C05497=1160.781,162.301,-57.931,-178.413,6.811,148.793
C05498=1160.776,162.550,-57.953,-178.410,6.813,148.793
C05499=1160.772,162.799,-57.975,-178.407,6.815,148.793
C05500=1160.767,163.048,-57.997,-178.404,6.817,148.792
C05501=1160.762,163.296,-58.018,-178.401,6.819,148.792
C05502=1160.758,163.546,-58.040,-178.399,6.821,148.792
C05503=1160.753,163.794,-58.062,-178.396,6.823,148.791
C05504=1160.749,164.044,-58.084,-178.394,6.824,148.791
C05505=1160.744,164.292,-58.106,-178.390,6.827,148.791
C05506=1160.740,164.542,-58.128,-178.388,6.829,148.790
C05507=1160.735,164.790,-58.149,-178.385,6.831,148.790
C05508=1160.731,165.040,-58.172,-178.382,6.832,148.790
C05509=1160.725,165.289,-58.194,-178.380,6.834,148.789
C05510=1160.721,165.538,-58.216,-178.377,6.836,148.789
C05511=1160.716,165.787,-58.238,-178.374,6.839,148.789
C05512=1160.712,166.036,-58.260,-178.371,6.840,148.788
C05513=1160.707,166.285,-58.281,-178.369,6.842,148.788
C05514=1160.703,166.534,-58.303,-178.366,6.844,148.788
C05515=1160.698,166.783,-58.325,-178.363,6.846,148.787
C05516=1160.692,167.032,-58.347,-178.360,6.848,148.787
C05517=1160.688,167.281,-58.369,-178.358,6.850,148.787
C05518=1160.683,167.529,-58.392,-178.355,6.852,148.786
C05519=1160.679,167.778,-58.414,-178.352,6.854,148.786
C05520=1160.675,168.028,-58.436,-178.350,6.856,148.786
C05521=1160.669,168.276,-58.458,-178.346,6.858,148.785
C05522=1160.665,168.526,-58.480,-178.344,6.860,148.785
C05523=1160.660,168.774,-58.502,-178.342,6.862,148.785
C05524=1160.656,169.023,-58.525,-178.339,6.864,148.784
C05525=1160.650,169.272,-58.547,-178.336,6.865,148.784
C05526=1160.646,169.521,-58.569,-178.333,6.868,148.784
C05527=1160.641,169.770,-58.591,-178.330,6.870,148.783
C05528=1160.637,170.019,-58.613,-178.328,6.872,148.783
C05529=1160.632,170.268,-58.636,-178.325,6.874,148.783
C05530=1160.627,170.517,-58.658,-178.322,6.876,148.782
C05531=1160.623,170.766,-58.679,-178.319,6.878,148.782
C05532=1160.618,171.015,-58.702,-178.317,6.880,148.782
C05533=1160.614,171.264,-58.725,-178.314,6.881,148.781
C05534=1160.609,171.513,-58.746,-178.312,6.884,148.781
C05535=1160.604,171.762,-58.769,-178.308,6.886,148.781
C05536=1160.599,172.010,-58.792,-178.306,6.888,148.780
C05537=1160.595,172.260,-58.814,-178.303,6.890,148.780
C05538=1160.590,172.509,-58.836,-178.300,6.891,148.780
C05539=1160.585,172.757,-58.859,-178.297,6.894,148.779
C05540=1160.581,173.007,-58.881,-178.295,6.896,148.779
C05541=1160.575,173.256,-58.903,-178.292,6.898,148.779
C05542=1160.571,173.504,-58.926,-178.290,6.899,148.779
C05543=1160.567,173.754,-58.948,-178.286,6.902,148.778
C05544=1160.562,174.002,-58.971,-178.284,6.904,148.778
C05545=1160.558,174.252,-58.993,-178.281,6.906,148.778
C05546=1160.553,174.501,-59.016,-178.279,6.908,148.777
C05547=1160.548,174.749,-59.038,-178.275,6.910,148.777
C05548=1160.544,174.998,-59.061,-178.273,6.912,148.777
C05549=1160.539,175.248,-59.083,-178.271,6.914,148.776
C05550=1160.534,175.496,-59.105,-178.268,6.916,148.776
C05551=1160.529,175.745,-59.128,-178.265,6.918,148.776
C05552=1160.525,175.995,-59.150,-178.262,6.920,148.775
C05553=1160.520,176.243,-59.173,-178.259,6.922,148.775
C05554=1160.516,176.492,-59.196,-178.256,6.925,148.775
C05555=1160.511,176.741,-59.219,-178.254,6.927,148.775
C05556=1160.506,176.989,-59.241,-178.251,6.928,148.774
C05557=1160.501,177.239,-59.264,-178.248,6.930,148.774
C05558=1160.497,177.488,-59.287,-178.246,6.933,148.774
C05559=1160.492,177.737,-59.309,-178.243,6.935,148.773
C05560=1160.488,177.985,-59.332,-178.240,6.936,148.773
C05561=1160.483,178.234,-59.355,-178.237,6.938,148.773
C05562=1160.479,178.484,-59.377,-178.235,6.941,148.772
C05563=1160.474,178.732,-59.400,-178.232,6.943,148.772
C05564=1160.470,178.981,-59.423,-178.229,6.945,148.772
C05565=1160.465,179.230,-59.445,-178.226,6.947,148.771
C05566=1160.461,179.479,-59.468,-178.224,6.949,148.771
C05567=1160.455,179.727,-59.491,-178.221,6.951,148.771
C05568=1160.450,179.977,-59.514,-178.218,6.953,148.771
C05569=1160.446,180.226,-59.537,-178.215,6.955,148.770
C05570=1160.442,180.475,-59.560,-178.213,6.958,148.770
C05571=1160.437,180.723,-59.582,-178.210,6.959,148.770
C05572=1160.432,180.973,-59.605,-178.207,6.962,148.769
C05573=1160.427,181.222,-59.628,-178.204,6.964,148.769
C05574=1160.423,181.470,-59.651,-178.202,6.966,148.769
C05575=1160.419,181.719,-59.674,-178.199,6.968,148.768
C05576=1160.414,181.968,-59.696,-178.196,6.970,148.768
C05577=1160.409,182.217,-59.719,-178.193,6.972,148.768
C05578=1160.404,182.466,-59.743,-178.191,6.975,148.768
C05579=1160.401,182.715,-59.766,-178.188,6.976,148.767
C05580=1160.396,182.964,-59.789,-178.185,6.978,148.767
C05581=1160.391,183.213,-59.812,-178.183,6.980,148.767
C05582=1160.386,183.461,-59.834,-178.180,6.983,148.766
C05583=1160.381,183.731,-59.860,-178.177,6.985,148.766
C05584=1160.376,184.000,-59.885,-178.174,6.987,148.766
C05585=1160.372,184.271,-59.910,-178.171,6.990,148.765
C05586=1160.367,184.540,-59.935,-178.168,6.992,148.765
C05587=1160.361,184.789,-59.958,-178.165,6.994,148.765
C05588=1160.357,185.038,-59.981,-178.162,6.996,148.765
C05589=1160.353,185.286,-60.004,-178.160,6.998,148.764
C05590=1160.348,185.535,-60.027,-178.157,7.001,148.764
C05591=1160.343,185.784,-60.050,-178.154,7.003,148.764
C05592=1160.339,186.033,-60.074,-178.152,7.004,148.763
C05593=1160.335,186.282,-60.097,-178.148,7.007,148.763
C05594=1160.330,186.531,-60.120,-178.146,7.009,148.763
C05595=1160.325,186.780,-60.143,-178.143,7.011,148.763
C05596=1160.320,187.029,-60.166,-178.140,7.013,148.762
C05597=1160.315,187.278,-60.190,-178.138,7.016,148.762
C05598=1160.311,187.526,-60.212,-178.135,7.017,148.762
C05599=1160.307,187.775,-60.236,-178.132,7.020,148.761
C05600=1160.302,188.024,-60.259,-178.130,7.022,148.761
C05601=1160.297,188.273,-60.282,-178.127,7.024,148.761
C05602=1160.292,188.522,-60.306,-178.124,7.026,148.761
C05603=1160.288,188.771,-60.330,-178.122,7.028,148.760
C05604=1160.283,189.020,-60.353,-178.119,7.030,148.760
C05605=1160.279,189.269,-60.377,-178.116,7.033,148.760
C05606=1160.275,189.518,-60.399,-178.114,7.035,148.760
C05607=1160.270,189.767,-60.423,-178.110,7.037,148.759
C05608=1160.265,190.015,-60.446,-178.108,7.039,148.759
C05609=1160.260,190.263,-60.470,-178.105,7.041,148.759
C05610=1160.256,190.512,-60.493,-178.102,7.044,148.758
C05611=1160.251,190.762,-60.517,-178.099,7.046,148.758
C05612=1160.246,191.011,-60.540,-178.097,7.048,148.758
C05613=1160.241,191.260,-60.563,-178.094,7.050,148.758
C05614=1160.237,191.508,-60.587,-178.091,7.052,148.757
C05615=1160.232,191.757,-60.611,-178.088,7.055,148.757
C05616=1160.228,192.006,-60.634,-178.086,7.057,148.757
C05617=1160.223,192.254,-60.658,-178.083,7.058,148.756
C05618=1160.219,192.504,-60.681,-178.080,7.061,148.756
C05619=1160.214,192.753,-60.705,-178.078,7.063,148.756
C05620=1160.210,193.001,-60.729,-178.075,7.065,148.756
C05621=1160.205,193.250,-60.752,-178.072,7.068,148.756
C05622=1160.200,193.499,-60.776,-178.069,7.070,148.755
C05623=1160.196,193.747,-60.800,-178.067,7.073,148.755
C05624=1160.191,193.996,-60.823,-178.064,7.074,148.755
C05625=1160.187,194.246,-60.847,-178.061,7.076,148.754
C05626=1160.183,194.495,-60.871,-178.059,7.079,148.754
C05627=1160.178,194.744,-60.894,-178.056,7.081,148.754
C05628=1160.173,194.992,-60.918,-178.053,7.083,148.754
C05629=1160.169,195.241,-60.942,-178.050,7.085,148.753
C05630=1160.164,195.490,-60.965,-178.047,7.088,148.753
C05631=1160.160,195.739,-60.989,-178.045,7.090,148.753
C05632=1160.155,195.988,-61.012,-178.042,7.092,148.753
C05633=1160.150,196.236,-61.037,-178.039,7.094,148.752
C05634=1160.145,196.485,-61.060,-178.037,7.097,148.752
C05635=1160.141,196.734,-61.085,-178.034,7.099,148.752
C05636=1160.136,196.983,-61.108,-178.031,7.101,148.752
C05637=1160.132,197.231,-61.132,-178.029,7.103,148.751
C05638=1160.128,197.480,-61.156,-178.025,7.106,148.751
C05639=1160.123,197.729,-61.180,-178.023,7.108,148.751
C05640=1160.119,197.978,-61.204,-178.020,7.110,148.751
C05641=1160.113,198.227,-61.228,-178.018,7.112,148.750
C05642=1160.109,198.475,-61.252,-178.014,7.115,148.750
C05643=1160.104,198.725,-61.275,-178.012,7.117,148.750
C05644=1160.100,198.973,-61.299,-178.010,7.119,148.750
C05645=1160.095,199.221,-61.323,-178.006,7.121,148.749
C05646=1160.091,199.471,-61.348,-178.004,7.124,148.749
C05647=1160.086,199.720,-61.372,-178.001,7.126,148.749
C05648=1160.082,199.968,-61.396,-177.998,7.128,148.749
C05649=1160.077,200.217,-61.419,-177.995,7.131,148.748
C05650=1160.073,200.466,-61.443,-177.993,7.133,148.748
C05651=1160.068,200.714,-61.468,-177.990,7.136,148.748
C05652=1160.063,200.964,-61.492,-177.987,7.137,148.748
C05653=1160.059,201.213,-61.516,-177.985,7.139,148.747
C05654=1160.055,201.461,-61.540,-177.982,7.142,148.747
C05655=1160.050,201.710,-61.565,-177.979,7.144,148.747
C05656=1160.045,201.959,-61.588,-177.976,7.147,148.747
C05657=1160.041,202.208,-61.612,-177.974,7.148,148.746
C05658=1160.036,202.457,-61.637,-177.971,7.151,148.746
C05659=1160.032,202.705,-61.661,-177.968,7.153,148.746
C05660=1160.027,202.953,-61.685,-177.965,7.156,148.746
C05661=1160.022,203.203,-61.709,-177.963,7.158,148.745
C05662=1160.018,203.452,-61.734,-177.960,7.161,148.745
C05663=1160.014,203.700,-61.758,-177.957,7.163,148.745
C05664=1160.008,203.949,-61.782,-177.954,7.165,148.745
C05665=1160.005,204.198,-61.807,-177.952,7.167,148.745
C05666=1160.000,204.446,-61.831,-177.949,7.169,148.744
C05667=1159.995,204.695,-61.855,-177.946,7.172,148.744
C05668=1159.991,204.944,-61.880,-177.944,7.174,148.744
C05669=1159.986,205.193,-61.905,-177.941,7.177,148.744
C05670=1159.981,205.442,-61.928,-177.938,7.178,148.743
C05671=1159.977,205.690,-61.952,-177.935,7.181,148.743
C05672=1159.972,205.939,-61.977,-177.933,7.183,148.743
C05673=1159.968,206.188,-62.001,-177.930,7.186,148.743
C05674=1159.963,206.437,-62.026,-177.927,7.188,148.742
C05675=1159.959,206.685,-62.050,-177.925,7.191,148.742
C05676=1159.954,206.935,-62.075,-177.922,7.192,148.742
C05677=1159.950,207.183,-62.099,-177.919,7.195,148.742
C05678=1159.945,207.432,-62.124,-177.916,7.197,148.742
C05679=1159.941,207.681,-62.148,-177.914,7.200,148.741
C05680=1159.936,207.929,-62.173,-177.911,7.202,148.741
C05681=1159.932,208.178,-62.198,-177.908,7.205,148.741
C05682=1159.926,208.426,-62.222,-177.905,7.207,148.741
C05683=1159.923,208.675,-62.247,-177.903,7.210,148.741
C05684=1159.917,208.924,-62.271,-177.900,7.211,148.740
C05685=1159.914,209.173,-62.296,-177.897,7.214,148.740
C05686=1159.909,209.422,-62.320,-177.895,7.216,148.740
C05687=1159.903,209.692,-62.347,-177.892,7.219,148.740
C05688=1159.899,209.963,-62.374,-177.889,7.221,148.739
C05689=1159.894,210.233,-62.401,-177.885,7.224,148.739
C05690=1159.889,210.504,-62.428,-177.882,7.227,148.739
C05691=1159.885,210.753,-62.452,-177.880,7.229,148.739
C05692=1159.880,211.001,-62.477,-177.877,7.232,148.739
C05693=1159.876,211.250,-62.501,-177.874,7.233,148.738
C05694=1159.871,211.498,-62.527,-177.872,7.236,148.738
C05695=1159.866,211.748,-62.552,-177.869,7.238,148.738
C05696=1159.862,211.996,-62.576,-177.866,7.241,148.738
C05697=1159.857,212.244,-62.601,-177.863,7.243,148.737
C05698=1159.853,212.494,-62.626,-177.861,7.246,148.737
C05699=1159.848,212.742,-62.650,-177.858,7.248,148.737
C05700=1159.844,212.992,-62.675,-177.855,7.251,148.737
C05701=1159.839,213.240,-62.701,-177.852,7.253,148.737
C05702=1159.835,213.488,-62.725,-177.850,7.255,148.736
C05703=1159.830,213.738,-62.750,-177.847,7.258,148.736
C05704=1159.825,213.986,-62.775,-177.844,7.260,148.736
C05705=1159.821,214.235,-62.800,-177.842,7.263,148.736
C05706=1159.817,214.483,-62.825,-177.839,7.265,148.735
C05707=1159.812,214.732,-62.850,-177.836,7.268,148.735
C05708=1159.808,214.981,-62.874,-177.833,7.269,148.735
C05709=1159.803,215.230,-62.900,-177.831,7.272,148.735
C05710=1159.798,215.478,-62.924,-177.828,7.275,148.735
C05711=1159.794,215.727,-62.950,-177.825,7.277,148.735
C05712=1159.790,215.976,-62.974,-177.822,7.280,148.734
C05713=1159.785,216.224,-63.000,-177.820,7.282,148.734
C05714=1159.780,216.473,-63.025,-177.817,7.285,148.734
C05715=1159.776,216.722,-63.050,-177.814,7.286,148.734
C05716=1159.772,216.970,-63.075,-177.812,7.289,148.734
C05717=1159.767,217.219,-63.100,-177.809,7.291,148.733
C05718=1159.762,217.468,-63.125,-177.806,7.294,148.733
C05719=1159.758,217.717,-63.151,-177.803,7.297,148.733
C05720=1159.753,217.965,-63.175,-177.801,7.299,148.733
C05721=1159.750,218.214,-63.201,-177.798,7.302,148.733
C05722=1159.744,218.463,-63.225,-177.795,7.303,148.732
C05723=1159.740,218.711,-63.251,-177.792,7.306,148.732
C05724=1159.736,218.960,-63.277,-177.790,7.309,148.732
C05725=1159.731,219.209,-63.301,-177.787,7.311,148.732
C05726=1159.727,219.458,-63.327,-177.784,7.314,148.732
C05727=1159.722,219.705,-63.352,-177.781,7.316,148.731
C05728=1159.718,219.955,-63.377,-177.779,7.319,148.731
C05729=1159.713,220.203,-63.402,-177.776,7.322,148.731
C05730=1159.709,220.452,-63.428,-177.773,7.323,148.731
C05731=1159.704,220.701,-63.453,-177.770,7.326,148.731
C05732=1159.700,220.949,-63.478,-177.768,7.328,148.730
C05733=1159.695,221.198,-63.504,-177.765,7.331,148.730
C05734=1159.690,221.446,-63.530,-177.762,7.334,148.730
C05735=1159.686,221.696,-63.555,-177.760,7.336,148.730
C05736=1159.682,221.944,-63.580,-177.757,7.339,148.730
C05737=1159.677,222.193,-63.606,-177.754,7.341,148.729
C05738=1159.673,222.441,-63.632,-177.751,7.343,148.729
C05739=1159.668,222.690,-63.656,-177.749,7.346,148.729
C05740=1159.663,222.939,-63.682,-177.746,7.348,148.729
C05741=1159.659,223.188,-63.708,-177.743,7.351,148.729
C05742=1159.654,223.436,-63.733,-177.741,7.353,148.729
C05743=1159.650,223.685,-63.759,-177.738,7.356,148.728
C05744=1159.646,223.933,-63.785,-177.735,7.359,148.728
C05745=1159.641,224.182,-63.809,-177.733,7.361,148.728
C05746=1159.636,224.431,-63.835,-177.729,7.363,148.728
C05747=1159.632,224.680,-63.861,-177.727,7.366,148.728
C05748=1159.627,224.928,-63.886,-177.724,7.368,148.728
C05749=1159.623,225.177,-63.912,-177.721,7.371,148.727
C05750=1159.619,225.425,-63.938,-177.718,7.374,148.727
C05751=1159.614,225.674,-63.963,-177.716,7.376,148.727
C05752=1159.610,225.922,-63.989,-177.713,7.379,148.727
C05753=1159.606,226.171,-64.015,-177.711,7.381,148.727
C05754=1159.601,226.420,-64.040,-177.708,7.383,148.727
C05755=1159.597,226.668,-64.066,-177.705,7.386,148.726
C05756=1159.592,226.917,-64.092,-177.703,7.389,148.726
C05757=1159.587,227.166,-64.118,-177.699,7.391,148.726
C05758=1159.583,227.414,-64.143,-177.697,7.394,148.726
C05759=1159.578,227.663,-64.169,-177.694,7.396,148.726
C05760=1159.574,227.912,-64.195,-177.691,7.399,148.726
C05761=1159.570,228.161,-64.220,-177.688,7.402,148.725
C05762=1159.565,228.409,-64.246,-177.686,7.404,148.725
C05763=1159.560,228.658,-64.272,-177.683,7.406,148.725
C05764=1159.556,228.906,-64.299,-177.680,7.409,148.725
C05765=1159.552,229.155,-64.324,-177.678,7.412,148.725
C05766=1159.547,229.403,-64.350,-177.675,7.414,148.725
C05767=1159.543,229.652,-64.375,-177.672,7.417,148.724
C05768=1159.538,229.901,-64.402,-177.670,7.419,148.724
C05769=1159.534,230.150,-64.428,-177.667,7.422,148.724
C05770=1159.530,230.398,-64.454,-177.664,7.425,148.724
C05771=1159.525,230.646,-64.479,-177.662,7.427,148.724
C05772=1159.520,230.895,-64.506,-177.659,7.430,148.724
C05773=1159.516,231.144,-64.532,-177.656,7.432,148.723
C05774=1159.512,231.393,-64.557,-177.653,7.434,148.723
C05775=1159.508,231.641,-64.584,-177.651,7.437,148.723
C05776=1159.502,231.889,-64.610,-177.648,7.440,148.723
C05777=1159.498,232.138,-64.635,-177.645,7.443,148.723
C05778=1159.494,232.386,-64.662,-177.642,7.445,148.723
C05779=1159.489,232.635,-64.688,-177.640,7.448,148.723
C05780=1159.485,232.884,-64.714,-177.636,7.451,148.722
C05781=1159.481,233.132,-64.741,-177.634,7.453,148.722
C05782=1159.475,233.381,-64.766,-177.631,7.456,148.722
C05783=1159.471,233.630,-64.792,-177.629,7.459,148.722
C05784=1159.467,233.878,-64.819,-177.626,7.460,148.722
C05785=1159.462,234.127,-64.845,-177.623,7.463,148.722
C05786=1159.458,234.376,-64.871,-177.620,7.466,148.722
C05787=1159.454,234.624,-64.897,-177.618,7.469,148.722
C05788=1159.449,234.873,-64.924,-177.615,7.471,148.721
C05789=1159.445,235.121,-64.950,-177.612,7.474,148.721
C05790=1159.440,235.370,-64.976,-177.609,7.477,148.721
C05791=1159.436,235.641,-65.005,-177.606,7.479,148.721
C05792=1159.431,235.913,-65.033,-177.603,7.482,148.721
C05793=1159.426,236.185,-65.063,-177.601,7.485,148.721
C05794=1159.421,236.457,-65.091,-177.597,7.488,148.720
C05795=1159.417,236.705,-65.118,-177.595,7.491,148.720
C05796=1159.413,236.954,-65.144,-177.592,7.493,148.720
C05797=1159.407,237.202,-65.170,-177.590,7.496,148.720
C05798=1159.403,237.450,-65.197,-177.586,7.499,148.720
C05799=1159.398,237.699,-65.223,-177.584,7.502,148.720
C05800=1159.394,237.947,-65.249,-177.581,7.504,148.720
C05801=1159.389,238.197,-65.276,-177.579,7.507,148.720
C05802=1159.386,238.445,-65.302,-177.576,7.510,148.719
C05803=1159.381,238.693,-65.329,-177.573,7.512,148.719
C05804=1159.377,238.942,-65.355,-177.570,7.514,148.719
C05805=1159.372,239.191,-65.382,-177.568,7.517,148.719
C05806=1159.368,239.439,-65.409,-177.565,7.520,148.719
C05807=1159.363,239.688,-65.435,-177.562,7.523,148.719
C05808=1159.358,239.936,-65.462,-177.559,7.525,148.718
C05809=1159.355,240.185,-65.488,-177.557,7.528,148.718
C05810=1159.350,240.434,-65.515,-177.554,7.531,148.718
C05811=1159.346,240.682,-65.541,-177.551,7.534,148.718
C05812=1159.341,240.930,-65.568,-177.548,7.535,148.718
C05813=1159.337,241.179,-65.595,-177.546,7.538,148.718
C05814=1159.332,241.428,-65.621,-177.543,7.541,148.718
C05815=1159.327,241.676,-65.648,-177.540,7.544,148.718
C05816=1159.324,241.924,-65.675,-177.538,7.546,148.718
C05817=1159.319,242.173,-65.702,-177.535,7.549,148.718
C05818=1159.314,242.421,-65.729,-177.532,7.552,148.717
C05819=1159.310,242.670,-65.755,-177.529,7.555,148.717
C05820=1159.305,242.919,-65.782,-177.527,7.557,148.717
C05821=1159.301,243.167,-65.809,-177.524,7.560,148.717
C05822=1159.297,243.415,-65.835,-177.521,7.563,148.717
C05823=1159.293,243.664,-65.863,-177.519,7.566,148.717
C05824=1159.288,243.913,-65.890,-177.515,7.568,148.717
C05825=1159.284,244.161,-65.916,-177.513,7.571,148.716
C05826=1159.279,244.410,-65.943,-177.510,7.574,148.716
C05827=1159.275,244.658,-65.970,-177.508,7.576,148.716
C05828=1159.271,244.907,-65.996,-177.505,7.579,148.716
C05829=1159.266,245.155,-66.023,-177.503,7.582,148.716
C05830=1159.261,245.404,-66.050,-177.500,7.584,148.716
C05831=1159.257,245.652,-66.077,-177.497,7.587,148.716
C05832=1159.253,245.901,-66.104,-177.494,7.590,148.716
C05833=1159.249,246.150,-66.131,-177.491,7.593,148.716
C05834=1159.244,246.398,-66.158,-177.489,7.595,148.716
C05835=1159.239,246.647,-66.185,-177.486,7.598,148.715
C05836=1159.235,246.895,-66.213,-177.483,7.601,148.715
C05837=1159.231,247.143,-66.239,-177.480,7.604,148.715
C05838=1159.226,247.391,-66.266,-177.477,7.607,148.715
C05839=1159.222,247.640,-66.294,-177.475,7.609,148.715
C05840=1159.218,247.889,-66.321,-177.473,7.612,148.715
C05841=1159.213,248.138,-66.348,-177.470,7.615,148.715
C05842=1159.208,248.386,-66.375,-177.467,7.618,148.715
C05843=1159.204,248.634,-66.402,-177.464,7.620,148.715
C05844=1159.200,248.883,-66.429,-177.462,7.623,148.715
C05845=1159.195,249.131,-66.456,-177.459,7.626,148.715
C05846=1159.191,249.380,-66.484,-177.456,7.628,148.714
C05847=1159.187,249.628,-66.511,-177.453,7.631,148.714
C05848=1159.182,249.877,-66.538,-177.450,7.634,148.714
C05849=1159.177,250.125,-66.565,-177.448,7.636,148.714
C05850=1159.173,250.373,-66.593,-177.446,7.639,148.714
C05851=1159.169,250.622,-66.620,-177.443,7.642,148.714
C05852=1159.164,250.871,-66.647,-177.440,7.645,148.714
C05853=1159.160,251.119,-66.674,-177.437,7.648,148.714
C05854=1159.156,251.367,-66.701,-177.434,7.651,148.714
C05855=1159.152,251.616,-66.729,-177.432,7.653,148.714
C05856=1159.147,251.865,-66.756,-177.429,7.656,148.714
C05857=1159.143,252.112,-66.784,-177.426,7.659,148.713
C05858=1159.138,252.361,-66.811,-177.423,7.662,148.713
C05859=1159.134,252.610,-66.838,-177.421,7.664,148.713
C05860=1159.130,252.858,-66.866,-177.418,7.667,148.713
C05861=1159.125,253.107,-66.893,-177.416,7.670,148.713
C05862=1159.121,253.354,-66.921,-177.413,7.672,148.713
C05863=1159.117,253.604,-66.948,-177.410,7.675,148.713
C05864=1159.112,253.852,-66.975,-177.407,7.678,148.713
C05865=1159.108,254.100,-67.003,-177.405,7.681,148.713
C05866=1159.104,254.349,-67.031,-177.402,7.684,148.713
C05867=1159.099,254.597,-67.059,-177.399,7.687,148.713
C05868=1159.094,254.846,-67.086,-177.397,7.689,148.712
C05869=1159.090,255.094,-67.114,-177.394,7.692,148.712
C05870=1159.086,255.343,-67.141,-177.391,7.695,148.712
C05871=1159.081,255.591,-67.169,-177.389,7.698,148.712
C05872=1159.077,255.839,-67.196,-177.386,7.701,148.712
C05873=1159.073,256.088,-67.224,-177.383,7.704,148.712
C05874=1159.068,256.336,-67.251,-177.381,7.706,148.712
C05875=1159.064,256.584,-67.279,-177.378,7.709,148.712
C05876=1159.059,256.834,-67.307,-177.375,7.712,148.712
C05877=1159.055,257.082,-67.335,-177.373,7.715,148.712
C05878=1159.051,257.330,-67.363,-177.370,7.718,148.712
C05879=1159.046,257.579,-67.390,-177.367,7.721,148.712
C05880=1159.042,257.827,-67.418,-177.364,7.724,148.711
C05881=1159.038,258.076,-67.445,-177.361,7.726,148.711
C05882=1159.033,258.324,-67.474,-177.359,7.729,148.711
C05883=1159.029,258.572,-67.501,-177.356,7.732,148.711
C05884=1159.025,258.820,-67.529,-177.353,7.735,148.711
C05885=1159.020,259.069,-67.557,-177.351,7.737,148.711
C05886=1159.016,259.318,-67.585,-177.348,7.740,148.711
C05887=1159.011,259.566,-67.613,-177.345,7.743,148.711
C05888=1159.007,259.814,-67.640,-177.342,7.746,148.711
C05889=1159.003,260.063,-67.668,-177.340,7.750,148.711
C05890=1158.999,260.311,-67.696,-177.338,7.752,148.711
C05891=1158.994,260.560,-67.725,-177.335,7.755,148.711
C05892=1158.989,260.808,-67.752,-177.332,7.758,148.711
C05893=1158.986,261.057,-67.780,-177.329,7.761,148.711
C05894=1158.981,261.304,-67.808,-177.327,7.763,148.711
C05895=1158.976,261.578,-67.839,-177.324,7.766,148.711
C05896=1158.971,261.851,-67.870,-177.320,7.770,148.710
C05897=1158.967,262.125,-67.900,-177.317,7.773,148.710
C05898=1158.962,262.398,-67.932,-177.315,7.776,148.710
C05899=1158.958,262.646,-67.959,-177.312,7.779,148.710
C05900=1158.953,262.895,-67.988,-177.309,7.782,148.710
C05901=1158.949,263.143,-68.015,-177.306,7.785,148.710
C05902=1158.944,263.392,-68.044,-177.304,7.788,148.710
C05903=1158.940,263.640,-68.072,-177.301,7.791,148.710
C05904=1158.936,263.888,-68.100,-177.298,7.794,148.710
C05905=1158.931,264.136,-68.128,-177.296,7.796,148.710
C05906=1158.927,264.385,-68.157,-177.294,7.799,148.710
C05907=1158.922,264.633,-68.185,-177.291,7.802,148.710
C05908=1158.918,264.882,-68.213,-177.288,7.805,148.710
C05909=1158.914,265.130,-68.241,-177.285,7.808,148.710
C05910=1158.910,265.378,-68.270,-177.282,7.811,148.710
C05911=1158.905,265.626,-68.297,-177.280,7.814,148.710
C05912=1158.901,265.875,-68.326,-177.277,7.817,148.710
C05913=1158.896,266.123,-68.354,-177.274,7.820,148.710
C05914=1158.892,266.372,-68.383,-177.271,7.822,148.710
C05915=1158.888,266.620,-68.410,-177.269,7.825,148.710
C05916=1158.883,266.868,-68.440,-177.266,7.829,148.710
C05917=1158.880,267.117,-68.468,-177.264,7.831,148.710
C05918=1158.875,267.365,-68.496,-177.261,7.834,148.710
C05919=1158.871,267.613,-68.524,-177.259,7.837,148.710
C05920=1158.866,267.862,-68.553,-177.256,7.840,148.709
C05921=1158.862,268.110,-68.581,-177.253,7.843,148.709
C05922=1158.857,268.358,-68.610,-177.250,7.846,148.709
C05923=1158.853,268.606,-68.638,-177.248,7.849,148.709
C05924=1158.849,268.855,-68.667,-177.245,7.851,148.709
C05925=1158.845,269.103,-68.695,-177.242,7.854,148.709
C05926=1158.840,269.352,-68.723,-177.240,7.858,148.709
C05927=1158.835,269.600,-68.753,-177.237,7.861,148.709
C05928=1158.832,269.848,-68.781,-177.234,7.864,148.709
C05929=1158.827,270.097,-68.809,-177.231,7.867,148.709
C05930=1158.823,270.344,-68.838,-177.229,7.870,148.709
C05931=1158.819,270.593,-68.867,-177.226,7.872,148.709
C05932=1158.814,270.842,-68.895,-177.223,7.875,148.709
C05933=1158.810,271.089,-68.924,-177.221,7.879,148.709
C05934=1158.806,271.338,-68.953,-177.219,7.881,148.709
C05935=1158.801,271.587,-68.981,-177.216,7.884,148.709
C05936=1158.797,271.834,-69.010,-177.213,7.887,148.709
C05937=1158.793,272.083,-69.039,-177.210,7.890,148.709
C05938=1158.788,272.332,-69.067,-177.208,7.893,148.709
C05939=1158.784,272.579,-69.096,-177.205,7.896,148.709
C05940=1158.779,272.828,-69.125,-177.203,7.899,148.709
C05941=1158.775,273.076,-69.154,-177.200,7.902,148.709
C05942=1158.771,273.324,-69.182,-177.197,7.905,148.709
C05943=1158.767,273.573,-69.211,-177.194,7.908,148.709
C05944=1158.762,273.822,-69.240,-177.191,7.911,148.709
C05945=1158.758,274.070,-69.269,-177.189,7.914,148.709
C05946=1158.754,274.318,-69.297,-177.186,7.917,148.709
C05947=1158.750,274.566,-69.327,-177.184,7.920,148.709
C05948=1158.745,274.815,-69.355,-177.181,7.923,148.709
C05949=1158.741,275.063,-69.385,-177.178,7.926,148.709
C05950=1158.737,275.311,-69.413,-177.175,7.929,148.709
C05951=1158.732,275.559,-69.442,-177.173,7.932,148.709
C05952=1158.728,275.807,-69.472,-177.170,7.935,148.709
C05953=1158.724,276.056,-69.500,-177.168,7.938,148.709
C05954=1158.719,276.304,-69.529,-177.165,7.941,148.709
C05955=1158.715,276.552,-69.558,-177.162,7.944,148.709
C05956=1158.711,276.801,-69.587,-177.160,7.947,148.709
C05957=1158.707,277.049,-69.616,-177.157,7.950,148.709
C05958=1158.702,277.297,-69.645,-177.154,7.953,148.709
C05959=1158.698,277.546,-69.674,-177.151,7.956,148.709
C05960=1158.693,277.794,-69.704,-177.149,7.959,148.709
C05961=1158.690,278.042,-69.733,-177.146,7.962,148.709
C05962=1158.685,278.291,-69.761,-177.144,7.965,148.709
C05963=1158.681,278.538,-69.790,-177.141,7.968,148.709
C05964=1158.676,278.786,-69.820,-177.138,7.971,148.709
C05965=1158.672,279.035,-69.849,-177.135,7.974,148.709
C05966=1158.668,279.284,-69.878,-177.133,7.977,148.709
C05967=1158.664,279.532,-69.908,-177.130,7.980,148.709
C05968=1158.659,279.780,-69.937,-177.127,7.983,148.709
C05969=1158.655,280.028,-69.966,-177.125,7.986,148.709
C05970=1158.650,280.276,-69.996,-177.122,7.989,148.709
C05971=1158.646,280.524,-70.025,-177.120,7.992,148.709
C05972=1158.642,280.773,-70.054,-177.117,7.995,148.709
C05973=1158.638,281.021,-70.083,-177.114,7.998,148.709
C05974=1158.633,281.270,-70.113,-177.112,8.002,148.709
C05975=1158.629,281.518,-70.142,-177.109,8.005,148.709
C05976=1158.625,281.766,-70.172,-177.106,8.007,148.709
C05977=1158.620,282.014,-70.201,-177.104,8.010,148.709
C05978=1158.616,282.262,-70.230,-177.101,8.014,148.709
C05979=1158.612,282.510,-70.260,-177.098,8.017,148.709
C05980=1158.608,282.759,-70.289,-177.096,8.020,148.709
C05981=1158.604,283.007,-70.318,-177.093,8.023,148.709
C05982=1158.599,283.255,-70.348,-177.091,8.026,148.709
C05983=1158.595,283.503,-70.377,-177.088,8.029,148.709
C05984=1158.591,283.752,-70.407,-177.085,8.032,148.709
C05985=1158.587,284.000,-70.436,-177.083,8.035,148.709
C05986=1158.583,284.248,-70.466,-177.080,8.038,148.709
C05987=1158.578,284.496,-70.495,-177.077,8.041,148.709
C05988=1158.574,284.744,-70.524,-177.075,8.044,148.709
C05989=1158.569,284.993,-70.554,-177.072,8.047,148.709
C05990=1158.565,285.241,-70.584,-177.069,8.050,148.709
C05991=1158.560,285.489,-70.613,-177.067,8.053,148.709
C05992=1158.557,285.737,-70.643,-177.064,8.056,148.709
C05993=1158.552,285.985,-70.673,-177.062,8.059,148.709
C05994=1158.548,286.233,-70.702,-177.059,8.062,148.709
C05995=1158.544,286.482,-70.732,-177.057,8.066,148.709
C05996=1158.539,286.730,-70.762,-177.054,8.069,148.709
C05997=1158.535,286.978,-70.791,-177.051,8.071,148.709
C05998=1158.531,287.226,-70.821,-177.049,8.075,148.709
C05999=1158.526,287.501,-70.854,-177.045,8.079,148.709
C06000=1158.521,287.776,-70.887,-177.043,8.081,148.709
C06001=1158.516,288.052,-70.920,-177.040,8.086,148.710
C06002=1158.512,288.326,-70.953,-177.037,8.089,148.710
C06003=1158.508,288.575,-70.983,-177.034,8.091,148.710
C06004=1158.504,288.824,-71.012,-177.031,8.096,148.710
C06005=1158.499,289.072,-71.043,-177.029,8.099,148.710
C06006=1158.495,289.320,-71.073,-177.026,8.102,148.710
C06007=1158.491,289.568,-71.102,-177.024,8.105,148.710
C06008=1158.486,289.816,-71.133,-177.021,8.108,148.710
C06009=1158.482,290.064,-71.162,-177.018,8.111,148.710
C06010=1158.478,290.312,-71.193,-177.016,8.114,148.710
C06011=1158.474,290.560,-71.222,-177.013,8.117,148.710
C06012=1158.469,290.809,-71.252,-177.010,8.120,148.710
C06013=1158.465,291.056,-71.282,-177.008,8.123,148.710
C06014=1158.461,291.305,-71.312,-177.005,8.126,148.710
C06015=1158.457,291.553,-71.342,-177.003,8.129,148.710
C06016=1158.452,291.801,-71.372,-177.000,8.132,148.710
C06017=1158.448,292.049,-71.403,-176.997,8.135,148.710
C06018=1158.444,292.298,-71.432,-176.995,8.139,148.710
C06019=1158.440,292.546,-71.463,-176.992,8.142,148.710
C06020=1158.435,292.794,-71.493,-176.989,8.145,148.710
C06021=1158.432,293.042,-71.523,-176.987,8.149,148.710
C06022=1158.427,293.290,-71.552,-176.984,8.152,148.710
C06023=1158.423,293.538,-71.583,-176.982,8.155,148.711
C06024=1158.419,293.786,-71.613,-176.979,8.158,148.711
C06025=1158.414,294.034,-71.643,-176.977,8.161,148.711
C06026=1158.411,294.283,-71.674,-176.974,8.164,148.711
C06027=1158.406,294.531,-71.704,-176.971,8.167,148.711
C06028=1158.402,294.779,-71.734,-176.969,8.170,148.711
C06029=1158.397,295.027,-71.765,-176.966,8.173,148.711
C06030=1158.393,295.275,-71.794,-176.964,8.177,148.711
C06031=1158.389,295.523,-71.824,-176.960,8.180,148.711
C06032=1158.385,295.771,-71.856,-176.958,8.183,148.711
C06033=1158.381,296.020,-71.885,-176.955,8.187,148.711
C06034=1158.376,296.268,-71.916,-176.952,8.190,148.711
C06035=1158.373,296.515,-71.946,-176.950,8.193,148.711
C06036=1158.368,296.764,-71.976,-176.947,8.196,148.711
C06037=1158.364,297.012,-72.007,-176.945,8.199,148.711
C06038=1158.360,297.260,-72.037,-176.942,8.202,148.711
C06039=1158.355,297.508,-72.068,-176.940,8.205,148.712
C06040=1158.351,297.756,-72.098,-176.937,8.208,148.712
C06041=1158.347,298.005,-72.129,-176.934,8.212,148.712
C06042=1158.343,298.253,-72.159,-176.932,8.215,148.712
C06043=1158.339,298.501,-72.190,-176.929,8.218,148.712
C06044=1158.334,298.749,-72.220,-176.927,8.222,148.712
C06045=1158.331,298.997,-72.251,-176.924,8.224,148.712
C06046=1158.326,299.245,-72.282,-176.922,8.228,148.712
C06047=1158.322,299.492,-72.312,-176.919,8.231,148.712
C06048=1158.317,299.741,-72.342,-176.916,8.234,148.712
C06049=1158.313,299.990,-72.373,-176.914,8.237,148.712
C06050=1158.309,300.237,-72.403,-176.911,8.241,148.712
C06051=1158.305,300.485,-72.434,-176.908,8.244,148.712
C06052=1158.300,300.733,-72.465,-176.906,8.247,148.713
C06053=1158.297,300.982,-72.495,-176.903,8.250,148.712
C06054=1158.292,301.230,-72.526,-176.901,8.254,148.713
C06055=1158.288,301.478,-72.557,-176.898,8.257,148.713
C06056=1158.284,301.726,-72.588,-176.896,8.260,148.713
C06057=1158.280,301.974,-72.618,-176.893,8.263,148.713
C06058=1158.275,302.222,-72.649,-176.890,8.267,148.713
C06059=1158.271,302.470,-72.680,-176.887,8.270,148.713
C06060=1158.266,302.718,-72.711,-176.885,8.273,148.713
C06061=1158.263,302.966,-72.741,-176.882,8.276,148.713
C06062=1158.259,303.214,-72.773,-176.880,8.279,148.713
C06063=1158.254,303.462,-72.803,-176.877,8.282,148.713
C06064=1158.250,303.710,-72.834,-176.875,8.286,148.713
C06065=1158.246,303.958,-72.865,-176.871,8.289,148.713
C06066=1158.242,304.206,-72.896,-176.869,8.293,148.714
C06067=1158.237,304.454,-72.926,-176.867,8.296,148.714
C06068=1158.233,304.703,-72.957,-176.864,8.299,148.714
C06069=1158.229,304.950,-72.989,-176.862,8.302,148.714
C06070=1158.224,305.198,-73.020,-176.859,8.305,148.714
C06071=1158.221,305.447,-73.050,-176.857,8.308,148.714
C06072=1158.216,305.695,-73.081,-176.853,8.312,148.714
C06073=1158.212,305.942,-73.112,-176.851,8.315,148.714
C06074=1158.208,306.191,-73.144,-176.848,8.318,148.714
C06075=1158.203,306.438,-73.174,-176.846,8.322,148.715
C06076=1158.199,306.687,-73.205,-176.844,8.325,148.715
C06077=1158.195,306.934,-73.237,-176.841,8.328,148.715
C06078=1158.191,307.183,-73.268,-176.839,8.331,148.715
C06079=1158.186,307.431,-73.299,-176.835,8.335,148.715
C06080=1158.183,307.678,-73.330,-176.833,8.338,148.715
C06081=1158.179,307.927,-73.361,-176.830,8.341,148.715
C06082=1158.174,308.175,-73.392,-176.828,8.345,148.715
C06083=1158.171,308.423,-73.423,-176.826,8.348,148.715
C06084=1158.166,308.671,-73.454,-176.823,8.351,148.715
C06085=1158.162,308.919,-73.486,-176.820,8.355,148.716
C06086=1158.158,309.167,-73.517,-176.817,8.358,148.716
C06087=1158.154,309.415,-73.548,-176.815,8.361,148.716
C06088=1158.149,309.663,-73.579,-176.813,8.364,148.716
C06089=1158.145,309.911,-73.611,-176.810,8.367,148.716
C06090=1158.141,310.159,-73.642,-176.807,8.371,148.716
C06091=1158.136,310.407,-73.673,-176.804,8.374,148.716
C06092=1158.133,310.655,-73.705,-176.802,8.378,148.716
C06093=1158.128,310.903,-73.735,-176.800,8.381,148.717
C06094=1158.124,311.151,-73.767,-176.797,8.384,148.716
C06095=1158.121,311.399,-73.799,-176.795,8.387,148.717
C06096=1158.116,311.647,-73.830,-176.792,8.391,148.717
C06097=1158.112,311.895,-73.862,-176.789,8.394,148.717
C06098=1158.107,312.143,-73.893,-176.787,8.398,148.717
C06099=1158.103,312.391,-73.925,-176.784,8.401,148.717
C06100=1158.099,312.639,-73.956,-176.782,8.404,148.717
C06101=1158.095,312.887,-73.988,-176.779,8.408,148.717
C06102=1158.091,313.134,-74.019,-176.776,8.411,148.717
C06103=1158.086,313.412,-74.055,-176.774,8.414,148.718
C06104=1158.081,313.689,-74.089,-176.771,8.418,148.718
C06105=1158.077,313.967,-74.125,-176.767,8.422,148.718
C06106=1158.072,314.244,-74.160,-176.765,8.426,148.718
C06107=1158.068,314.492,-74.192,-176.762,8.429,148.718
C06108=1158.064,314.740,-74.223,-176.759,8.432,148.718
C06109=1158.060,314.988,-74.254,-176.757,8.436,148.718
C06110=1158.055,315.236,-74.287,-176.755,8.439,148.719
C06111=1158.051,315.483,-74.318,-176.752,8.443,148.719
C06112=1158.047,315.731,-74.350,-176.749,8.446,148.719
C06113=1158.043,315.980,-74.381,-176.747,8.449,148.719
C06114=1158.039,316.227,-74.413,-176.744,8.452,148.719
C06115=1158.035,316.476,-74.445,-176.742,8.456,148.719
C06116=1158.030,316.723,-74.477,-176.739,8.460,148.719
C06117=1158.027,316.971,-74.509,-176.736,8.463,148.719
C06118=1158.023,317.219,-74.540,-176.734,8.466,148.720
C06119=1158.018,317.467,-74.573,-176.732,8.469,148.720
C06120=1158.014,317.716,-74.604,-176.729,8.473,148.720
C06121=1158.010,317.964,-74.635,-176.726,8.476,148.720
C06122=1158.006,318.211,-74.667,-176.724,8.480,148.720
C06123=1158.001,318.459,-74.699,-176.721,8.483,148.720
C06124=1157.998,318.707,-74.731,-176.719,8.486,148.721
C06125=1157.993,318.955,-74.763,-176.716,8.490,148.721
C06126=1157.989,319.203,-74.795,-176.713,8.493,148.721
C06127=1157.985,319.451,-74.827,-176.711,8.496,148.721
C06128=1157.981,319.698,-74.859,-176.708,8.499,148.721
C06129=1157.976,319.947,-74.891,-176.705,8.504,148.721
C06130=1157.973,320.195,-74.923,-176.703,8.507,148.721
C06131=1157.969,320.443,-74.955,-176.701,8.510,148.722
C06132=1157.964,320.690,-74.987,-176.698,8.513,148.722
C06133=1157.961,320.938,-75.019,-176.695,8.517,148.722
C06134=1157.957,321.186,-75.051,-176.693,8.520,148.722
C06135=1157.952,321.434,-75.084,-176.691,8.524,148.722
C06136=1157.948,321.682,-75.115,-176.688,8.527,148.722
C06137=1157.944,321.930,-75.147,-176.685,8.531,148.723
C06138=1157.940,322.178,-75.179,-176.683,8.534,148.723
C06139=1157.936,322.426,-75.211,-176.680,8.537,148.723
C06140=1157.932,322.673,-75.244,-176.678,8.541,148.723
C06141=1157.928,322.921,-75.276,-176.675,8.544,148.723
C06142=1157.923,323.169,-75.308,-176.672,8.548,148.723
C06143=1157.920,323.417,-75.340,-176.670,8.551,148.724
C06144=1157.915,323.665,-75.373,-176.668,8.554,148.724
C06145=1157.911,323.913,-75.405,-176.665,8.558,148.724
C06146=1157.907,324.161,-75.437,-176.662,8.561,148.724
C06147=1157.903,324.409,-75.469,-176.660,8.565,148.724
C06148=1157.899,324.657,-75.502,-176.658,8.568,148.724
C06149=1157.895,324.904,-75.534,-176.655,8.572,148.725
C06150=1157.890,325.152,-75.566,-176.652,8.575,148.725
C06151=1157.887,325.400,-75.599,-176.650,8.578,148.725
C06152=1157.882,325.648,-75.631,-176.647,8.582,148.725
C06153=1157.879,325.896,-75.663,-176.644,8.586,148.725
C06154=1157.875,326.144,-75.696,-176.642,8.589,148.725
C06155=1157.869,326.392,-75.728,-176.640,8.592,148.726
C06156=1157.866,326.639,-75.761,-176.636,8.596,148.726
C06157=1157.862,326.887,-75.793,-176.634,8.599,148.726
C06158=1157.858,327.135,-75.826,-176.632,8.603,148.726
C06159=1157.854,327.383,-75.858,-176.630,8.606,148.726
C06160=1157.849,327.631,-75.891,-176.627,8.610,148.726
C06161=1157.846,327.879,-75.923,-176.624,8.613,148.727
C06162=1157.841,328.127,-75.955,-176.622,8.616,148.727
C06163=1157.837,328.374,-75.988,-176.619,8.620,148.727
C06164=1157.833,328.622,-76.020,-176.616,8.624,148.727
C06165=1157.829,328.870,-76.053,-176.614,8.627,148.727
C06166=1157.825,329.118,-76.087,-176.612,8.630,148.727
C06167=1157.821,329.366,-76.118,-176.609,8.634,148.728
C06168=1157.817,329.613,-76.152,-176.607,8.637,148.728
C06169=1157.812,329.862,-76.184,-176.604,8.641,148.728
C06170=1157.809,330.109,-76.217,-176.601,8.645,148.728
C06171=1157.805,330.357,-76.250,-176.599,8.648,148.728
C06172=1157.800,330.605,-76.282,-176.596,8.651,148.729
C06173=1157.796,330.852,-76.315,-176.594,8.654,148.729
C06174=1157.792,331.100,-76.347,-176.591,8.658,148.729
C06175=1157.788,331.348,-76.380,-176.589,8.662,148.729
C06176=1157.784,331.596,-76.413,-176.587,8.665,148.729
C06177=1157.780,331.844,-76.446,-176.584,8.669,148.730
C06178=1157.776,332.092,-76.478,-176.581,8.672,148.730
C06179=1157.772,332.339,-76.511,-176.579,8.676,148.730
C06180=1157.768,332.587,-76.544,-176.576,8.680,148.730
C06181=1157.764,332.835,-76.578,-176.573,8.683,148.730
C06182=1157.759,333.083,-76.610,-176.571,8.686,148.730
C06183=1157.756,333.331,-76.643,-176.568,8.690,148.731
C06184=1157.752,333.578,-76.676,-176.566,8.693,148.731
C06185=1157.747,333.826,-76.709,-176.564,8.697,148.731
C06186=1157.743,334.074,-76.742,-176.561,8.701,148.731
C06187=1157.739,334.322,-76.774,-176.558,8.704,148.732
C06188=1157.735,334.570,-76.808,-176.556,8.707,148.732
C06189=1157.731,334.818,-76.841,-176.553,8.712,148.732
C06190=1157.726,335.065,-76.874,-176.551,8.715,148.732
C06191=1157.723,335.313,-76.907,-176.549,8.718,148.732
C06192=1157.719,335.560,-76.940,-176.546,8.722,148.733
C06193=1157.715,335.808,-76.973,-176.543,8.725,148.733
C06194=1157.711,336.056,-77.006,-176.541,8.729,148.733
C06195=1157.706,336.304,-77.039,-176.538,8.733,148.733
C06196=1157.702,336.551,-77.072,-176.536,8.736,148.734
C06197=1157.698,336.799,-77.105,-176.534,8.739,148.734
C06198=1157.694,337.047,-77.139,-176.531,8.744,148.734
C06199=1157.691,337.295,-77.172,-176.528,8.747,148.734
C06200=1157.686,337.543,-77.205,-176.526,8.750,148.734
C06201=1157.682,337.791,-77.238,-176.523,8.754,148.735
C06202=1157.678,338.038,-77.272,-176.521,8.757,148.735
C06203=1157.674,338.286,-77.305,-176.519,8.761,148.735
C06204=1157.670,338.534,-77.338,-176.516,8.765,148.735
C06205=1157.666,338.782,-77.371,-176.513,8.768,148.735
C06206=1157.662,339.029,-77.404,-176.511,8.771,148.736
C06207=1157.657,339.309,-77.442,-176.508,8.776,148.736
C06208=1157.653,339.589,-77.480,-176.505,8.780,148.736
C06209=1157.648,339.869,-77.517,-176.502,8.784,148.736
C06210=1157.643,340.149,-77.555,-176.500,8.788,148.737
C06211=1157.639,340.396,-77.588,-176.497,8.792,148.737
C06212=1157.635,340.645,-77.622,-176.494,8.795,148.737
C06213=1157.632,340.892,-77.656,-176.492,8.798,148.737
C06214=1157.627,341.140,-77.689,-176.489,8.803,148.738
C06215=1157.623,341.387,-77.722,-176.487,8.806,148.738
C06216=1157.619,341.635,-77.755,-176.485,8.809,148.738
C06217=1157.615,341.882,-77.789,-176.482,8.813,148.738
C06218=1157.610,342.130,-77.823,-176.479,8.817,148.738
C06219=1157.607,342.379,-77.856,-176.476,8.821,148.739
C06220=1157.603,342.626,-77.890,-176.474,8.824,148.739
C06221=1157.599,342.874,-77.923,-176.472,8.827,148.739
C06222=1157.595,343.121,-77.957,-176.469,8.832,148.740
C06223=1157.590,343.369,-77.991,-176.467,8.835,148.740
C06224=1157.587,343.617,-78.025,-176.464,8.839,148.740
C06225=1157.582,343.865,-78.058,-176.462,8.842,148.740
C06226=1157.579,344.112,-78.092,-176.460,8.846,148.740
C06227=1157.575,344.360,-78.125,-176.457,8.850,148.741
C06228=1157.570,344.607,-78.159,-176.454,8.853,148.741
C06229=1157.566,344.856,-78.193,-176.451,8.857,148.741
C06230=1157.563,345.103,-78.227,-176.449,8.860,148.741
C06231=1157.558,345.350,-78.260,-176.447,8.864,148.742
C06232=1157.554,345.598,-78.294,-176.444,8.868,148.742
C06233=1157.550,345.846,-78.328,-176.442,8.871,148.742
C06234=1157.547,346.093,-78.362,-176.439,8.875,148.743
C06235=1157.542,346.341,-78.395,-176.437,8.879,148.743
C06236=1157.538,346.589,-78.429,-176.435,8.882,148.743
C06237=1157.534,346.837,-78.463,-176.432,8.886,148.743
C06238=1157.530,347.084,-78.497,-176.429,8.889,148.743
C06239=1157.526,347.332,-78.531,-176.426,8.893,148.744
C06240=1157.522,347.580,-78.565,-176.425,8.897,148.744
C06241=1157.518,347.827,-78.599,-176.422,8.901,148.744
C06242=1157.514,348.075,-78.632,-176.419,8.904,148.745
C06243=1157.510,348.322,-78.666,-176.417,8.908,148.745
C06244=1157.506,348.570,-78.701,-176.414,8.912,148.745
C06245=1157.502,348.818,-78.734,-176.412,8.915,148.745
C06246=1157.498,349.065,-78.768,-176.409,8.920,148.746
C06247=1157.494,349.313,-78.803,-176.407,8.923,148.746
C06248=1157.490,349.560,-78.837,-176.404,8.927,148.746
C06249=1157.485,349.808,-78.870,-176.402,8.930,148.746
C06250=1157.482,350.056,-78.905,-176.400,8.933,148.747
C06251=1157.477,350.304,-78.939,-176.397,8.938,148.747
C06252=1157.474,350.551,-78.973,-176.395,8.941,148.747
C06253=1157.470,350.799,-79.007,-176.392,8.945,148.747
C06254=1157.465,351.047,-79.041,-176.390,8.949,148.748
C06255=1157.462,351.294,-79.075,-176.387,8.953,148.748
C06256=1157.458,351.542,-79.110,-176.384,8.956,148.748
C06257=1157.454,351.789,-79.144,-176.382,8.960,148.749
C06258=1157.450,352.037,-79.178,-176.380,8.964,148.749
C06259=1157.446,352.284,-79.212,-176.377,8.968,148.749
C06260=1157.442,352.533,-79.246,-176.375,8.971,148.749
C06261=1157.438,352.780,-79.280,-176.373,8.975,148.750
C06262=1157.433,353.027,-79.315,-176.370,8.979,148.750
C06263=1157.430,353.275,-79.349,-176.367,8.982,148.750
C06264=1157.426,353.523,-79.383,-176.365,8.986,148.750
C06265=1157.422,353.771,-79.418,-176.363,8.990,148.751
C06266=1157.418,354.018,-79.452,-176.360,8.994,148.751
C06267=1157.413,354.265,-79.487,-176.357,8.997,148.751
C06268=1157.410,354.513,-79.521,-176.355,9.001,148.752
C06269=1157.405,354.761,-79.555,-176.353,9.005,148.752
C06270=1157.402,355.008,-79.590,-176.350,9.009,148.752
C06271=1157.398,355.256,-79.624,-176.348,9.012,148.753
C06272=1157.394,355.504,-79.659,-176.345,9.016,148.753
C06273=1157.390,355.751,-79.693,-176.343,9.020,148.753
C06274=1157.386,355.999,-79.728,-176.340,9.024,148.753
C06275=1157.382,356.246,-79.763,-176.338,9.027,148.754
C06276=1157.378,356.494,-79.797,-176.335,9.032,148.754
C06277=1157.374,356.741,-79.831,-176.333,9.035,148.754
C06278=1157.370,356.989,-79.866,-176.330,9.039,148.755
C06279=1157.366,357.236,-79.900,-176.328,9.043,148.755
C06280=1157.362,357.484,-79.936,-176.325,9.047,148.755
C06281=1157.358,357.731,-79.970,-176.323,9.050,148.756
C06282=1157.354,357.979,-80.004,-176.320,9.054,148.756
C06283=1157.350,358.227,-80.039,-176.318,9.058,148.756
C06284=1157.346,358.475,-80.074,-176.315,9.062,148.756
C06285=1157.342,358.721,-80.109,-176.313,9.065,148.757
C06286=1157.338,358.969,-80.143,-176.310,9.069,148.757
C06287=1157.334,359.217,-80.178,-176.308,9.073,148.757
C06288=1157.330,359.464,-80.213,-176.305,9.077,148.758
C06289=1157.326,359.712,-80.248,-176.303,9.081,148.758
C06290=1157.322,359.959,-80.282,-176.300,9.085,148.758
C06291=1157.319,360.207,-80.317,-176.298,9.089,148.759
C06292=1157.314,360.454,-80.352,-176.296,9.092,148.759
C06293=1157.310,360.702,-80.387,-176.293,9.096,148.759
C06294=1157.307,360.950,-80.422,-176.290,9.100,148.759
C06295=1157.303,361.197,-80.456,-176.288,9.104,148.760
C06296=1157.299,361.445,-80.492,-176.285,9.108,148.760
C06297=1157.294,361.692,-80.526,-176.283,9.112,148.761
C06298=1157.291,361.940,-80.562,-176.280,9.116,148.761
C06299=1157.287,362.188,-80.597,-176.278,9.119,148.761
C06300=1157.283,362.435,-80.630,-176.276,9.124,148.762
C06301=1157.279,362.682,-80.666,-176.273,9.127,148.762
C06302=1157.275,362.930,-80.701,-176.271,9.131,148.762
C06303=1157.271,363.177,-80.736,-176.268,9.135,148.763
C06304=1157.267,363.425,-80.772,-176.266,9.139,148.763
C06305=1157.263,363.673,-80.806,-176.263,9.143,148.763
C06306=1157.259,363.920,-80.842,-176.261,9.146,148.763
C06307=1157.255,364.168,-80.876,-176.258,9.151,148.764
C06308=1157.252,364.415,-80.912,-176.255,9.155,148.764
C06309=1157.247,364.662,-80.947,-176.254,9.158,148.765
C06310=1157.243,364.910,-80.982,-176.251,9.162,148.765
C06311=1157.239,365.192,-81.022,-176.248,9.167,148.765
C06312=1157.235,365.476,-81.063,-176.246,9.171,148.766
C06313=1157.230,365.758,-81.102,-176.242,9.176,148.766
C06314=1157.225,366.041,-81.143,-176.240,9.181,148.767
C06315=1157.222,366.288,-81.178,-176.238,9.184,148.767
C06316=1157.218,366.536,-81.213,-176.235,9.188,148.767
C06317=1157.213,366.783,-81.248,-176.233,9.193,148.768
C06318=1157.210,367.031,-81.284,-176.230,9.196,148.768
C06319=1157.206,367.278,-81.319,-176.228,9.200,148.769
C06320=1157.202,367.526,-81.354,-176.226,9.204,148.769
C06321=1157.198,367.773,-81.389,-176.223,9.208,148.769
C06322=1157.194,368.021,-81.425,-176.221,9.212,148.770
C06323=1157.191,368.268,-81.461,-176.219,9.216,148.770
C06324=1157.187,368.516,-81.496,-176.216,9.221,148.771
C06325=1157.183,368.762,-81.531,-176.214,9.224,148.771
C06326=1157.179,369.011,-81.566,-176.211,9.228,148.771
C06327=1157.174,369.258,-81.602,-176.210,9.232,148.772
C06328=1157.171,369.506,-81.638,-176.207,9.236,148.772
C06329=1157.166,369.753,-81.673,-176.205,9.240,148.773
C06330=1157.163,370.000,-81.709,-176.203,9.244,148.773
C06331=1157.159,370.248,-81.744,-176.201,9.248,148.773
C06332=1157.155,370.495,-81.780,-176.198,9.252,148.774
C06333=1157.152,370.743,-81.815,-176.197,9.256,148.774
C06334=1157.147,370.990,-81.851,-176.194,9.260,148.775
C06335=1157.143,371.237,-81.886,-176.192,9.264,148.775
C06336=1157.139,371.485,-81.922,-176.190,9.268,148.776
C06337=1157.136,371.732,-81.958,-176.188,9.272,148.776
C06338=1157.132,371.980,-81.993,-176.186,9.275,148.777
C06339=1157.128,372.228,-82.029,-176.184,9.280,148.777
C06340=1157.123,372.474,-82.064,-176.182,9.284,148.778
C06341=1157.120,372.722,-82.100,-176.180,9.288,148.778
C06342=1157.116,372.969,-82.136,-176.178,9.292,148.779
C06343=1157.112,373.217,-82.171,-176.176,9.295,148.779
C06344=1157.108,373.464,-82.208,-176.174,9.300,148.780
C06345=1157.105,373.712,-82.244,-176.172,9.304,148.780
C06346=1157.101,373.959,-82.279,-176.170,9.307,148.781
C06347=1157.096,374.206,-82.315,-176.168,9.312,148.781
C06348=1157.092,374.454,-82.350,-176.166,9.315,148.782
C06349=1157.089,374.701,-82.386,-176.165,9.319,148.782
C06350=1157.085,374.948,-82.422,-176.162,9.324,148.783
C06351=1157.081,375.196,-82.458,-176.161,9.328,148.783
C06352=1157.077,375.443,-82.494,-176.159,9.332,148.784
C06353=1157.074,375.691,-82.529,-176.157,9.335,148.784
C06354=1157.069,375.938,-82.566,-176.156,9.339,148.785
C06355=1157.066,376.186,-82.602,-176.154,9.344,148.786
C06356=1157.062,376.433,-82.637,-176.152,9.347,148.786
C06357=1157.057,376.680,-82.673,-176.151,9.351,148.787
C06358=1157.054,376.927,-82.709,-176.149,9.355,148.787
C06359=1157.049,377.175,-82.746,-176.148,9.359,148.788
C06360=1157.046,377.422,-82.781,-176.146,9.363,148.789
C06361=1157.042,377.669,-82.817,-176.145,9.367,148.789
C06362=1157.038,377.917,-82.854,-176.143,9.371,148.790
C06363=1157.034,378.165,-82.889,-176.142,9.375,148.790
C06364=1157.030,378.412,-82.926,-176.140,9.379,148.791
C06365=1157.027,378.659,-82.961,-176.139,9.382,148.792
C06366=1157.023,378.906,-82.998,-176.137,9.386,148.792
C06367=1157.019,379.154,-83.034,-176.136,9.390,148.793
C06368=1157.015,379.402,-83.069,-176.135,9.394,148.794
C06369=1157.011,379.649,-83.106,-176.134,9.398,148.794
C06370=1157.007,379.896,-83.142,-176.133,9.401,148.795
C06371=1157.003,380.143,-83.179,-176.131,9.405,148.796
C06372=1157.000,380.391,-83.214,-176.130,9.410,148.796
C06373=1156.996,380.638,-83.251,-176.129,9.413,148.797
C06374=1156.992,380.886,-83.287,-176.128,9.417,148.798
C06375=1156.988,381.133,-83.323,-176.127,9.421,148.798
C06376=1156.984,381.380,-83.359,-176.126,9.425,148.799
C06377=1156.980,381.627,-83.396,-176.125,9.428,148.800
C06378=1156.976,381.875,-83.431,-176.124,9.432,148.801
C06379=1156.972,382.122,-83.468,-176.123,9.435,148.801
C06380=1156.969,382.370,-83.504,-176.122,9.439,148.802
C06381=1156.964,382.617,-83.541,-176.122,9.443,148.803
C06382=1156.961,382.864,-83.576,-176.120,9.447,148.804
C06383=1156.957,383.112,-83.613,-176.120,9.450,148.804
C06384=1156.953,383.359,-83.649,-176.119,9.454,148.805
C06385=1156.949,383.606,-83.686,-176.118,9.458,148.806
C06386=1156.946,383.853,-83.722,-176.118,9.461,148.806
C06387=1156.941,384.101,-83.758,-176.117,9.464,148.807
C06388=1156.938,384.348,-83.794,-176.117,9.468,148.808
C06389=1156.933,384.596,-83.830,-176.116,9.471,148.809
C06390=1156.930,384.842,-83.867,-176.116,9.475,148.810
C06391=1156.926,385.090,-83.903,-176.115,9.478,148.810
C06392=1156.922,385.337,-83.940,-176.115,9.481,148.811
C06393=1156.918,385.584,-83.976,-176.114,9.485,148.812
C06394=1156.914,385.832,-84.013,-176.114,9.489,148.813
C06395=1156.910,386.079,-84.048,-176.114,9.492,148.814
C06396=1156.906,386.326,-84.085,-176.114,9.495,148.814
C06397=1156.902,386.573,-84.122,-176.113,9.499,148.815
C06398=1156.899,386.821,-84.158,-176.114,9.502,148.816
C06399=1156.895,387.068,-84.194,-176.113,9.505,148.817
C06400=1156.892,387.316,-84.231,-176.113,9.509,148.818
C06401=1156.887,387.564,-84.267,-176.113,9.511,148.818
C06402=1156.883,387.811,-84.304,-176.113,9.515,148.819
C06403=1156.880,388.058,-84.340,-176.113,9.517,148.820
C06404=1156.876,388.305,-84.377,-176.113,9.521,148.821
C06405=1156.872,388.552,-84.413,-176.113,9.524,148.822
C06406=1156.868,388.799,-84.450,-176.114,9.526,148.822
C06407=1156.864,389.047,-84.486,-176.114,9.530,148.823
C06408=1156.861,389.294,-84.523,-176.114,9.533,148.824
C06409=1156.856,389.541,-84.559,-176.114,9.535,148.825
C06410=1156.852,389.789,-84.596,-176.114,9.538,148.826
C06411=1156.849,390.035,-84.632,-176.114,9.542,148.827
C06412=1156.845,390.283,-84.669,-176.115,9.545,148.828
C06413=1156.842,390.531,-84.705,-176.115,9.547,148.828
C06414=1156.838,390.778,-84.742,-176.116,9.550,148.829
C06415=1156.833,391.063,-84.784,-176.116,9.553,148.830
C06416=1156.829,391.349,-84.826,-176.117,9.556,148.831
C06417=1156.824,391.636,-84.868,-176.117,9.559,148.832
C06418=1156.819,391.921,-84.911,-176.118,9.563,148.833
C06419=1156.815,392.169,-84.948,-176.118,9.565,148.834
C06420=1156.812,392.416,-84.983,-176.118,9.568,148.835
C06421=1156.808,392.663,-85.020,-176.119,9.571,148.836
C06422=1156.805,392.911,-85.057,-176.120,9.573,148.836
C06423=1156.801,393.158,-85.093,-176.120,9.576,148.837
C06424=1156.797,393.405,-85.130,-176.121,9.578,148.838
C06425=1156.793,393.653,-85.166,-176.121,9.581,148.839
C06426=1156.789,393.900,-85.203,-176.122,9.583,148.840
C06427=1156.785,394.147,-85.240,-176.122,9.586,148.840
C06428=1156.781,394.394,-85.276,-176.123,9.588,148.841
C06429=1156.777,394.641,-85.313,-176.124,9.591,148.842
C06430=1156.773,394.888,-85.350,-176.124,9.593,148.843
C06431=1156.769,395.136,-85.386,-176.125,9.595,148.844
C06432=1156.766,395.384,-85.422,-176.125,9.598,148.844
C06433=1156.762,395.631,-85.459,-176.127,9.600,148.845
C06434=1156.758,395.878,-85.496,-176.127,9.603,148.846
C06435=1156.755,396.125,-85.532,-176.128,9.605,148.847
C06436=1156.750,396.373,-85.568,-176.128,9.608,148.848
C06437=1156.746,396.620,-85.605,-176.129,9.609,148.848
C06438=1156.743,396.867,-85.642,-176.130,9.612,148.849
C06439=1156.739,397.114,-85.678,-176.131,9.614,148.850
C06440=1156.735,397.361,-85.715,-176.131,9.616,148.851
C06441=1156.731,397.609,-85.753,-176.132,9.619,148.852
C06442=1156.728,397.856,-85.789,-176.133,9.621,148.853
C06443=1156.723,398.104,-85.825,-176.133,9.624,148.853
C06444=1156.719,398.351,-85.862,-176.134,9.626,148.854
C06445=1156.716,398.598,-85.898,-176.135,9.627,148.855
C06446=1156.712,398.845,-85.935,-176.136,9.629,148.856
C06447=1156.708,399.092,-85.972,-176.136,9.632,148.856
C06448=1156.704,399.340,-86.009,-176.137,9.634,148.857
C06449=1156.700,399.588,-86.045,-176.138,9.636,148.858
C06450=1156.696,399.835,-86.081,-176.139,9.638,148.859
C06451=1156.692,400.082,-86.118,-176.140,9.641,148.860
C06452=1156.689,400.329,-86.155,-176.140,9.642,148.860
C06453=1156.685,400.576,-86.191,-176.142,9.644,148.861
C06454=1156.681,400.823,-86.228,-176.142,9.646,148.862
C06455=1156.677,401.070,-86.265,-176.143,9.648,148.863
C06456=1156.673,401.318,-86.301,-176.143,9.651,148.863
C06457=1156.669,401.565,-86.338,-176.145,9.653,148.864
C06458=1156.665,401.813,-86.375,-176.145,9.655,148.865
C06459=1156.662,402.060,-86.411,-176.146,9.656,148.865
C06460=1156.658,402.307,-86.448,-176.147,9.658,148.866
C06461=1156.654,402.554,-86.485,-176.148,9.660,148.867
C06462=1156.650,402.802,-86.522,-176.149,9.662,148.868
C06463=1156.646,403.048,-86.558,-176.149,9.665,148.868
C06464=1156.642,403.296,-86.594,-176.150,9.667,148.869
C06465=1156.638,403.543,-86.631,-176.151,9.669,148.870
C06466=1156.635,403.791,-86.667,-176.152,9.670,148.871
C06467=1156.631,404.038,-86.704,-176.152,9.672,148.871
C06468=1156.627,404.285,-86.741,-176.153,9.674,148.872
C06469=1156.623,404.533,-86.778,-176.154,9.676,148.873
C06470=1156.620,404.779,-86.814,-176.155,9.678,148.873
C06471=1156.615,405.027,-86.851,-176.156,9.680,148.874
C06472=1156.611,405.275,-86.887,-176.157,9.682,148.875
C06473=1156.608,405.522,-86.924,-176.157,9.683,148.875
C06474=1156.604,405.769,-86.961,-176.158,9.685,148.876
C06475=1156.600,406.016,-86.998,-176.159,9.687,148.877
C06476=1156.596,406.264,-87.035,-176.160,9.689,148.878
C06477=1156.593,406.511,-87.071,-176.160,9.691,148.878
C06478=1156.589,406.758,-87.108,-176.161,9.693,148.879
C06479=1156.584,407.005,-87.144,-176.161,9.695,148.880
C06480=1156.580,407.252,-87.181,-176.162,9.697,148.880
C06481=1156.577,407.500,-87.217,-176.163,9.699,148.881
C06482=1156.573,407.748,-87.254,-176.164,9.700,148.882
C06483=1156.569,407.995,-87.291,-176.164,9.702,148.882
C06484=1156.566,408.242,-87.327,-176.165,9.704,148.883
C06485=1156.562,408.489,-87.364,-176.166,9.706,148.884
C06486=1156.558,408.736,-87.401,-176.166,9.707,148.884
C06487=1156.553,408.983,-87.438,-176.168,9.710,148.885
C06488=1156.551,409.231,-87.474,-176.168,9.711,148.886
C06489=1156.547,409.478,-87.511,-176.169,9.713,148.886
C06490=1156.543,409.725,-87.548,-176.170,9.715,148.887
C06491=1156.538,409.973,-87.584,-176.170,9.716,148.888
C06492=1156.535,410.220,-87.621,-176.171,9.718,148.888
C06493=1156.531,410.467,-87.657,-176.172,9.720,148.889
C06494=1156.527,410.714,-87.694,-176.172,9.722,148.890
C06495=1156.522,410.961,-87.731,-176.173,9.724,148.890
C06496=1156.520,411.209,-87.768,-176.173,9.726,148.891
C06497=1156.516,411.456,-87.805,-176.174,9.728,148.892
C06498=1156.512,411.703,-87.841,-176.175,9.730,148.892
C06499=1156.507,411.951,-87.878,-176.175,9.731,148.893
C06500=1156.504,412.197,-87.915,-176.176,9.733,148.894
C06501=1156.500,412.445,-87.951,-176.177,9.735,148.894
C06502=1156.496,412.692,-87.988,-176.177,9.736,148.895
C06503=1156.492,412.940,-88.025,-176.178,9.738,148.895
C06504=1156.489,413.187,-88.061,-176.178,9.740,148.896
C06505=1156.485,413.434,-88.098,-176.179,9.741,148.897
C06506=1156.481,413.682,-88.135,-176.179,9.744,148.897
C06507=1156.476,413.929,-88.172,-176.180,9.746,148.898
C06508=1156.473,414.176,-88.208,-176.180,9.748,148.899
C06509=1156.469,414.423,-88.245,-176.181,9.749,148.899
C06510=1156.465,414.671,-88.282,-176.181,9.751,148.900
C06511=1156.461,414.918,-88.319,-176.182,9.752,148.900
C06512=1156.458,415.165,-88.355,-176.183,9.754,148.901
C06513=1156.455,415.412,-88.392,-176.183,9.756,148.902
C06514=1156.454,415.659,-88.429,-176.184,9.759,148.902
C06515=1156.452,416.052,-88.486,-176.185,9.761,148.903
C06516=1156.454,416.444,-88.543,-176.185,9.764,148.904
C06517=1156.456,416.837,-88.601,-176.186,9.766,148.905
C06518=1156.461,417.228,-88.658,-176.187,9.768,148.906
C06519=1156.041,417.230,-88.705,-176.189,9.780,148.909
C06520=1156.036,416.835,-88.647,-176.189,9.777,148.909
C06521=1156.033,416.440,-88.590,-176.188,9.775,148.908
C06522=1156.032,416.044,-88.532,-176.187,9.771,148.907
C06523=1156.033,415.648,-88.474,-176.186,9.769,148.906
C06524=1156.035,415.401,-88.437,-176.186,9.768,148.905
C06525=1156.038,415.154,-88.400,-176.185,9.765,148.904
C06526=1156.041,414.906,-88.364,-176.185,9.764,148.904
C06527=1156.045,414.659,-88.327,-176.185,9.762,148.903
C06528=1156.048,414.412,-88.291,-176.184,9.760,148.903
C06529=1156.052,414.165,-88.254,-176.183,9.758,148.902
C06530=1156.056,413.918,-88.217,-176.182,9.757,148.901
C06531=1156.060,413.670,-88.180,-176.182,9.755,148.901
C06532=1156.063,413.422,-88.144,-176.181,9.753,148.900
C06533=1156.068,413.175,-88.107,-176.181,9.750,148.899
C06534=1156.072,412.928,-88.070,-176.180,9.749,148.899
C06535=1156.076,412.681,-88.034,-176.180,9.747,148.898
C06536=1156.080,412.434,-87.997,-176.179,9.745,148.898
C06537=1156.083,412.187,-87.960,-176.179,9.744,148.897
C06538=1156.087,411.939,-87.923,-176.178,9.742,148.896
C06539=1156.091,411.692,-87.886,-176.177,9.740,148.896
C06540=1156.095,411.444,-87.849,-176.177,9.739,148.895
C06541=1156.098,411.198,-87.813,-176.176,9.737,148.894
C06542=1156.102,410.950,-87.776,-176.175,9.735,148.894
C06543=1156.106,410.703,-87.740,-176.175,9.733,148.893
C06544=1156.110,410.456,-87.703,-176.174,9.732,148.893
C06545=1156.114,410.208,-87.667,-176.173,9.730,148.892
C06546=1156.118,409.961,-87.630,-176.173,9.727,148.891
C06547=1156.122,409.713,-87.593,-176.172,9.725,148.891
C06548=1156.126,409.466,-87.556,-176.171,9.723,148.890
C06549=1156.129,409.219,-87.520,-176.171,9.722,148.889
C06550=1156.133,408.972,-87.483,-176.170,9.720,148.888
C06551=1156.137,408.725,-87.446,-176.169,9.718,148.888
C06552=1156.140,408.477,-87.410,-176.169,9.716,148.887
C06553=1156.144,408.230,-87.373,-176.168,9.715,148.886
C06554=1156.148,407.983,-87.336,-176.167,9.713,148.886
C06555=1156.152,407.736,-87.299,-176.166,9.711,148.885
C06556=1156.156,407.489,-87.263,-176.166,9.709,148.885
C06557=1156.160,407.241,-87.227,-176.165,9.707,148.884
C06558=1156.164,406.994,-87.190,-176.164,9.706,148.883
C06559=1156.168,406.746,-87.152,-176.163,9.704,148.882
C06560=1156.171,406.499,-87.116,-176.163,9.702,148.882
C06561=1156.175,406.252,-87.079,-176.162,9.700,148.881
C06562=1156.179,406.005,-87.043,-176.161,9.698,148.880
C06563=1156.183,405.758,-87.006,-176.160,9.697,148.880
C06564=1156.187,405.511,-86.969,-176.159,9.695,148.879
C06565=1156.191,405.263,-86.933,-176.158,9.693,148.878
C06566=1156.195,405.016,-86.896,-176.158,9.691,148.878
C06567=1156.198,404.768,-86.860,-176.157,9.689,148.877
C06568=1156.202,404.521,-86.823,-176.157,9.687,148.876
C06569=1156.206,404.274,-86.786,-176.156,9.685,148.875
C06570=1156.210,404.027,-86.749,-176.155,9.683,148.875
C06571=1156.214,403.780,-86.713,-176.154,9.681,148.874
C06572=1156.218,403.532,-86.676,-176.153,9.679,148.873
C06573=1156.222,403.285,-86.639,-176.152,9.677,148.873
C06574=1156.225,403.037,-86.602,-176.151,9.675,148.872
C06575=1156.229,402.790,-86.566,-176.151,9.673,148.871
C06576=1156.233,402.543,-86.530,-176.150,9.672,148.870
C06577=1156.237,402.295,-86.493,-176.149,9.670,148.870
C06578=1156.241,402.049,-86.456,-176.148,9.668,148.869
C06579=1156.245,401.801,-86.420,-176.148,9.665,148.868
C06580=1156.249,401.554,-86.383,-176.147,9.663,148.867
C06581=1156.253,401.307,-86.346,-176.146,9.661,148.867
C06582=1156.256,401.059,-86.309,-176.145,9.659,148.866
C06583=1156.260,400.812,-86.272,-176.144,9.657,148.865
C06584=1156.264,400.564,-86.236,-176.143,9.656,148.864
C06585=1156.268,400.317,-86.199,-176.142,9.654,148.864
C06586=1156.272,400.070,-86.163,-176.142,9.651,148.863
C06587=1156.276,399.823,-86.126,-176.141,9.649,148.862
C06588=1156.280,399.576,-86.089,-176.140,9.647,148.861
C06589=1156.283,399.329,-86.053,-176.139,9.645,148.861
C06590=1156.287,399.081,-86.016,-176.139,9.643,148.860
C06591=1156.291,398.834,-85.979,-176.138,9.641,148.859
C06592=1156.295,398.586,-85.943,-176.137,9.639,148.858
C06593=1156.298,398.339,-85.907,-176.136,9.637,148.857
C06594=1156.303,398.092,-85.870,-176.135,9.634,148.857
C06595=1156.307,397.845,-85.833,-176.135,9.632,148.856
C06596=1156.310,397.598,-85.797,-176.134,9.630,148.855
C06597=1156.314,397.351,-85.760,-176.133,9.627,148.854
C06598=1156.318,397.103,-85.723,-176.132,9.625,148.854
C06599=1156.322,396.855,-85.686,-176.131,9.623,148.853
C06600=1156.325,396.608,-85.650,-176.131,9.621,148.852
C06601=1156.329,396.361,-85.613,-176.130,9.619,148.851
C06602=1156.333,396.114,-85.576,-176.130,9.616,148.850
C06603=1156.337,395.867,-85.540,-176.128,9.614,148.849
C06604=1156.341,395.620,-85.503,-176.128,9.611,148.849
C06605=1156.345,395.373,-85.466,-176.127,9.609,148.848
C06606=1156.349,395.125,-85.431,-176.127,9.606,148.847
C06607=1156.352,394.877,-85.394,-176.126,9.605,148.846
C06608=1156.356,394.630,-85.357,-176.125,9.602,148.845
C06609=1156.360,394.383,-85.320,-176.124,9.600,148.845
C06610=1156.364,394.136,-85.284,-176.124,9.597,148.844
C06611=1156.368,393.889,-85.247,-176.124,9.594,148.843
C06612=1156.372,393.641,-85.211,-176.122,9.592,148.842
C06613=1156.376,393.394,-85.174,-176.122,9.589,148.841
C06614=1156.380,393.147,-85.138,-176.122,9.587,148.841
C06615=1156.384,392.900,-85.101,-176.121,9.584,148.840
C06616=1156.387,392.652,-85.064,-176.120,9.582,148.839
C06617=1156.391,392.404,-85.028,-176.120,9.579,148.838
C06618=1156.395,392.157,-84.991,-176.119,9.576,148.837
C06619=1156.398,391.910,-84.955,-176.119,9.573,148.836
C06620=1156.403,391.625,-84.912,-176.118,9.571,148.835
C06621=1156.407,391.338,-84.870,-176.118,9.568,148.834
C06622=1156.412,391.052,-84.828,-176.118,9.564,148.834
C06623=1156.416,390.767,-84.786,-176.117,9.561,148.832
C06624=1156.420,390.519,-84.748,-176.117,9.558,148.832
C06625=1156.424,390.271,-84.712,-176.116,9.555,148.831
C06626=1156.428,390.024,-84.676,-176.116,9.553,148.830
C06627=1156.432,389.777,-84.639,-176.116,9.550,148.829
C06628=1156.435,389.530,-84.603,-176.116,9.546,148.828
C06629=1156.440,389.282,-84.567,-176.115,9.544,148.828
C06630=1156.444,389.035,-84.530,-176.115,9.541,148.827
C06631=1156.447,388.788,-84.494,-176.115,9.538,148.826
C06632=1156.451,388.541,-84.457,-176.115,9.535,148.825
C06633=1156.456,388.293,-84.421,-176.115,9.532,148.824
C06634=1156.459,388.046,-84.384,-176.115,9.528,148.823
C06635=1156.462,387.799,-84.347,-176.115,9.526,148.823
C06636=1156.466,387.552,-84.311,-176.115,9.522,148.822
C06637=1156.470,387.304,-84.275,-176.115,9.519,148.821
C06638=1156.474,387.057,-84.238,-176.115,9.516,148.820
C06639=1156.478,386.810,-84.202,-176.114,9.513,148.819
C06640=1156.482,386.562,-84.166,-176.115,9.510,148.818
C06641=1156.486,386.315,-84.129,-176.115,9.506,148.818
C06642=1156.489,386.068,-84.092,-176.115,9.503,148.817
C06643=1156.494,385.821,-84.056,-176.115,9.500,148.816
C06644=1156.497,385.573,-84.020,-176.116,9.497,148.815
C06645=1156.501,385.326,-83.983,-176.116,9.493,148.815
C06646=1156.505,385.079,-83.947,-176.116,9.490,148.814
C06647=1156.509,384.831,-83.911,-176.117,9.486,148.813
C06648=1156.513,384.584,-83.874,-176.117,9.483,148.812
C06649=1156.517,384.337,-83.838,-176.118,9.480,148.811
C06650=1156.520,384.089,-83.801,-176.119,9.475,148.810
C06651=1156.524,383.842,-83.765,-176.119,9.472,148.810
C06652=1156.528,383.594,-83.729,-176.119,9.469,148.809
C06653=1156.531,383.347,-83.692,-176.120,9.465,148.808
C06654=1156.535,383.100,-83.656,-176.121,9.461,148.808
C06655=1156.539,382.853,-83.620,-176.122,9.458,148.807
C06656=1156.543,382.605,-83.583,-176.122,9.455,148.806
C06657=1156.548,382.358,-83.547,-176.123,9.450,148.805
C06658=1156.551,382.111,-83.511,-176.124,9.447,148.805
C06659=1156.555,381.863,-83.475,-176.125,9.443,148.804
C06660=1156.559,381.616,-83.438,-176.126,9.440,148.803
C06661=1156.563,381.368,-83.402,-176.127,9.436,148.802
C06662=1156.567,381.121,-83.366,-176.128,9.432,148.802
C06663=1156.571,380.873,-83.330,-176.129,9.429,148.801
C06664=1156.574,380.627,-83.294,-176.130,9.424,148.800
C06665=1156.579,380.379,-83.257,-176.132,9.420,148.800
C06666=1156.582,380.132,-83.221,-176.133,9.417,148.799
C06667=1156.586,379.884,-83.185,-176.133,9.413,148.798
C06668=1156.590,379.637,-83.149,-176.135,9.409,148.798
C06669=1156.593,379.390,-83.113,-176.136,9.405,148.797
C06670=1156.598,379.143,-83.076,-176.137,9.401,148.796
C06671=1156.601,378.895,-83.041,-176.139,9.397,148.796
C06672=1156.605,378.648,-83.004,-176.140,9.393,148.795
C06673=1156.609,378.400,-82.968,-176.142,9.389,148.794
C06674=1156.614,378.153,-82.933,-176.143,9.386,148.794
C06675=1156.617,377.906,-82.896,-176.145,9.382,148.793
C06676=1156.621,377.659,-82.861,-176.146,9.378,148.792
C06677=1156.625,377.411,-82.825,-176.148,9.374,148.792
C06678=1156.629,377.164,-82.788,-176.149,9.370,148.791
C06679=1156.633,376.916,-82.752,-176.151,9.366,148.791
C06680=1156.637,376.669,-82.717,-176.152,9.362,148.790
C06681=1156.640,376.422,-82.680,-176.154,9.359,148.790
C06682=1156.645,376.174,-82.644,-176.155,9.355,148.789
C06683=1156.648,375.927,-82.609,-176.157,9.350,148.788
C06684=1156.652,375.680,-82.572,-176.159,9.346,148.788
C06685=1156.656,375.432,-82.536,-176.161,9.342,148.787
C06686=1156.660,375.184,-82.501,-176.162,9.339,148.787
C06687=1156.664,374.938,-82.466,-176.165,9.334,148.786
C06688=1156.668,374.690,-82.429,-176.166,9.330,148.785
C06689=1156.672,374.443,-82.393,-176.168,9.327,148.785
C06690=1156.675,374.195,-82.358,-176.169,9.323,148.784
C06691=1156.680,373.948,-82.322,-176.172,9.318,148.784
C06692=1156.683,373.700,-82.286,-176.174,9.315,148.784
C06693=1156.687,373.453,-82.250,-176.176,9.310,148.783
C06694=1156.690,373.206,-82.214,-176.178,9.306,148.782
C06695=1156.695,372.959,-82.178,-176.180,9.303,148.782
C06696=1156.699,372.711,-82.143,-176.182,9.298,148.781
C06697=1156.703,372.464,-82.107,-176.184,9.295,148.781
C06698=1156.706,372.216,-82.072,-176.186,9.290,148.780
C06699=1156.711,371.968,-82.036,-176.188,9.287,148.780
C06700=1156.714,371.721,-82.000,-176.190,9.283,148.780
C06701=1156.718,371.473,-81.964,-176.192,9.279,148.779
C06702=1156.722,371.227,-81.929,-176.194,9.275,148.779
C06703=1156.726,370.979,-81.894,-176.197,9.271,148.778
C06704=1156.730,370.731,-81.858,-176.198,9.267,148.778
C06705=1156.734,370.484,-81.822,-176.201,9.263,148.777
C06706=1156.738,370.236,-81.787,-176.203,9.259,148.777
C06707=1156.742,369.989,-81.751,-176.205,9.255,148.776
C06708=1156.746,369.742,-81.716,-176.207,9.251,148.776
C06709=1156.749,369.494,-81.680,-176.210,9.247,148.776
C06710=1156.754,369.247,-81.644,-176.211,9.243,148.775
C06711=1156.757,368.999,-81.609,-176.214,9.239,148.775
C06712=1156.762,368.752,-81.573,-176.216,9.235,148.774
C06713=1156.765,368.505,-81.538,-176.219,9.231,148.774
C06714=1156.769,368.257,-81.503,-176.221,9.227,148.773
C06715=1156.773,368.009,-81.467,-176.223,9.223,148.773
C06716=1156.777,367.762,-81.432,-176.226,9.219,148.773
C06717=1156.781,367.515,-81.397,-176.228,9.215,148.772
C06718=1156.785,367.267,-81.361,-176.230,9.211,148.772
C06719=1156.788,367.020,-81.326,-176.232,9.207,148.771
C06720=1156.793,366.772,-81.291,-176.235,9.203,148.771
C06721=1156.796,366.525,-81.256,-176.238,9.199,148.771
C06722=1156.801,366.277,-81.219,-176.239,9.195,148.770
C06723=1156.805,366.030,-81.184,-176.242,9.191,148.770
C06724=1156.809,365.747,-81.145,-176.245,9.187,148.770
C06725=1156.814,365.464,-81.104,-176.248,9.183,148.769
C06726=1156.818,365.181,-81.064,-176.251,9.177,148.769
C06727=1156.823,364.898,-81.024,-176.253,9.173,148.768
C06728=1156.826,364.651,-80.988,-176.256,9.169,148.768
C06729=1156.831,364.404,-80.953,-176.258,9.165,148.768
C06730=1156.835,364.156,-80.918,-176.261,9.161,148.767
C06731=1156.838,363.909,-80.883,-176.263,9.158,148.767
C06732=1156.842,363.661,-80.849,-176.266,9.153,148.767
C06733=1156.846,363.414,-80.813,-176.268,9.149,148.766
C06734=1156.850,363.166,-80.778,-176.270,9.146,148.766
C06735=1156.854,362.919,-80.743,-176.273,9.142,148.766
C06736=1156.858,362.671,-80.708,-176.275,9.138,148.765
C06737=1156.862,362.423,-80.673,-176.278,9.134,148.765
C06738=1156.866,362.176,-80.638,-176.280,9.130,148.765
C06739=1156.870,361.928,-80.603,-176.283,9.126,148.764
C06740=1156.873,361.681,-80.568,-176.286,9.122,148.764
C06741=1156.877,361.434,-80.533,-176.288,9.119,148.764
C06742=1156.881,361.186,-80.499,-176.290,9.114,148.763
C06743=1156.886,360.939,-80.463,-176.293,9.110,148.763
C06744=1156.890,360.691,-80.429,-176.295,9.107,148.763
C06745=1156.893,360.443,-80.394,-176.298,9.103,148.762
C06746=1156.897,360.196,-80.359,-176.300,9.099,148.762
C06747=1156.901,359.948,-80.324,-176.303,9.095,148.762
C06748=1156.905,359.701,-80.289,-176.305,9.092,148.761
C06749=1156.909,359.453,-80.254,-176.308,9.088,148.761
C06750=1156.913,359.206,-80.220,-176.311,9.083,148.761
C06751=1156.917,358.958,-80.185,-176.313,9.080,148.761
C06752=1156.921,358.710,-80.150,-176.316,9.076,148.760
C06753=1156.925,358.463,-80.116,-176.318,9.072,148.760
C06754=1156.928,358.216,-80.081,-176.321,9.068,148.760
C06755=1156.933,357.968,-80.046,-176.323,9.065,148.759
C06756=1156.937,357.720,-80.011,-176.325,9.060,148.759
C06757=1156.941,357.473,-79.977,-176.328,9.057,148.759
C06758=1156.944,357.226,-79.942,-176.331,9.053,148.758
C06759=1156.949,356.978,-79.907,-176.332,9.049,148.758
C06760=1156.953,356.730,-79.873,-176.335,9.045,148.758
C06761=1156.957,356.483,-79.839,-176.338,9.042,148.758
C06762=1156.961,356.235,-79.804,-176.340,9.038,148.757
C06763=1156.965,355.988,-79.770,-176.342,9.034,148.757
C06764=1156.969,355.740,-79.735,-176.345,9.030,148.757
C06765=1156.973,355.493,-79.700,-176.348,9.027,148.756
C06766=1156.976,355.245,-79.666,-176.350,9.023,148.756
C06767=1156.981,354.997,-79.631,-176.352,9.019,148.756
C06768=1156.985,354.749,-79.597,-176.355,9.015,148.755
C06769=1156.988,354.502,-79.563,-176.357,9.012,148.755
C06770=1156.992,354.254,-79.528,-176.360,9.007,148.755
C06771=1156.996,354.007,-79.494,-176.362,9.004,148.755
C06772=1157.001,353.760,-79.459,-176.365,9.000,148.754
C06773=1157.005,353.511,-79.425,-176.367,8.997,148.754
C06774=1157.009,353.264,-79.391,-176.370,8.992,148.754
C06775=1157.013,353.016,-79.356,-176.372,8.989,148.753
C06776=1157.016,352.769,-79.322,-176.375,8.985,148.753
C06777=1157.020,352.521,-79.287,-176.377,8.981,148.753
C06778=1157.024,352.274,-79.253,-176.380,8.977,148.752
C06779=1157.029,352.026,-79.220,-176.382,8.974,148.752
C06780=1157.032,351.778,-79.185,-176.385,8.970,148.752
C06781=1157.037,351.531,-79.151,-176.387,8.966,148.752
C06782=1157.040,351.283,-79.117,-176.389,8.963,148.751
C06783=1157.045,351.035,-79.082,-176.392,8.959,148.751
C06784=1157.048,350.788,-79.048,-176.395,8.956,148.751
C06785=1157.052,350.540,-79.013,-176.397,8.952,148.751
C06786=1157.057,350.292,-78.980,-176.399,8.948,148.750
C06787=1157.061,350.045,-78.946,-176.402,8.944,148.750
C06788=1157.064,349.797,-78.912,-176.404,8.941,148.750
C06789=1157.068,349.550,-78.878,-176.407,8.937,148.749
C06790=1157.073,349.302,-78.844,-176.410,8.933,148.749
C06791=1157.076,349.054,-78.810,-176.412,8.930,148.749
C06792=1157.081,348.807,-78.775,-176.414,8.926,148.749
C06793=1157.085,348.559,-78.742,-176.417,8.922,148.748
C06794=1157.088,348.311,-78.708,-176.420,8.918,148.748
C06795=1157.093,348.064,-78.673,-176.422,8.915,148.748
C06796=1157.097,347.816,-78.640,-176.425,8.911,148.748
C06797=1157.100,347.568,-78.606,-176.427,8.907,148.747
C06798=1157.105,347.321,-78.572,-176.430,8.903,148.747
C06799=1157.109,347.073,-78.538,-176.432,8.900,148.747
C06800=1157.113,346.825,-78.504,-176.434,8.897,148.747
C06801=1157.117,346.578,-78.470,-176.437,8.892,148.746
C06802=1157.121,346.330,-78.437,-176.439,8.889,148.746
C06803=1157.125,346.083,-78.403,-176.442,8.885,148.746
C06804=1157.129,345.834,-78.369,-176.445,8.882,148.746
C06805=1157.133,345.587,-78.335,-176.447,8.878,148.745
C06806=1157.137,345.340,-78.302,-176.449,8.874,148.745
C06807=1157.141,345.092,-78.267,-176.452,8.871,148.745
C06808=1157.145,344.844,-78.234,-176.455,8.867,148.745
C06809=1157.149,344.597,-78.200,-176.457,8.863,148.744
C06810=1157.153,344.349,-78.167,-176.460,8.859,148.744
C06811=1157.158,344.101,-78.132,-176.462,8.856,148.744
C06812=1157.162,343.854,-78.099,-176.464,8.853,148.744
C06813=1157.165,343.605,-78.065,-176.467,8.849,148.743
C06814=1157.169,343.358,-78.032,-176.469,8.845,148.743
C06815=1157.173,343.110,-77.998,-176.472,8.841,148.743
C06816=1157.178,342.862,-77.965,-176.474,8.838,148.743
C06817=1157.182,342.615,-77.931,-176.477,8.834,148.742
C06818=1157.185,342.367,-77.897,-176.480,8.830,148.742
C06819=1157.190,342.119,-77.864,-176.482,8.827,148.742
C06820=1157.193,341.872,-77.830,-176.485,8.823,148.742
C06821=1157.198,341.624,-77.796,-176.487,8.820,148.741
C06822=1157.202,341.376,-77.763,-176.489,8.816,148.741
C06823=1157.206,341.129,-77.729,-176.492,8.812,148.741
C06824=1157.210,340.881,-77.696,-176.495,8.809,148.741
C06825=1157.214,340.633,-77.663,-176.497,8.806,148.741
C06826=1157.218,340.385,-77.630,-176.500,8.802,148.740
C06827=1157.222,340.138,-77.596,-176.502,8.798,148.740
C06828=1157.228,339.858,-77.558,-176.505,8.794,148.740
C06829=1157.232,339.577,-77.520,-176.507,8.790,148.739
C06830=1157.236,339.298,-77.483,-176.510,8.786,148.739
C06831=1157.241,339.018,-77.445,-176.513,8.782,148.739
C06832=1157.245,338.770,-77.412,-176.516,8.778,148.739
C06833=1157.249,338.523,-77.379,-176.518,8.774,148.738
C06834=1157.253,338.276,-77.345,-176.521,8.771,148.738
C06835=1157.256,338.027,-77.312,-176.523,8.768,148.738
C06836=1157.261,337.779,-77.278,-176.526,8.764,148.738
C06837=1157.265,337.532,-77.245,-176.528,8.760,148.738
C06838=1157.269,337.284,-77.212,-176.531,8.757,148.737
C06839=1157.273,337.036,-77.179,-176.533,8.753,148.737
C06840=1157.277,336.789,-77.146,-176.536,8.750,148.737
C06841=1157.281,336.541,-77.113,-176.539,8.745,148.737
C06842=1157.285,336.293,-77.080,-176.541,8.742,148.736
C06843=1157.289,336.045,-77.046,-176.543,8.739,148.736
C06844=1157.294,335.798,-77.013,-176.546,8.735,148.736
C06845=1157.298,335.550,-76.980,-176.548,8.732,148.736
C06846=1157.302,335.302,-76.947,-176.551,8.729,148.736
C06847=1157.306,335.054,-76.914,-176.554,8.724,148.736
C06848=1157.309,334.807,-76.881,-176.556,8.721,148.735
C06849=1157.314,334.559,-76.849,-176.559,8.718,148.735
C06850=1157.318,334.311,-76.816,-176.562,8.714,148.735
C06851=1157.322,334.063,-76.782,-176.564,8.711,148.735
C06852=1157.326,333.815,-76.749,-176.566,8.707,148.735
C06853=1157.330,333.568,-76.716,-176.569,8.703,148.734
C06854=1157.335,333.320,-76.683,-176.571,8.700,148.734
C06855=1157.338,333.072,-76.651,-176.574,8.697,148.734
C06856=1157.342,332.824,-76.618,-176.577,8.692,148.734
C06857=1157.347,332.577,-76.585,-176.579,8.689,148.733
C06858=1157.351,332.329,-76.552,-176.581,8.686,148.733
C06859=1157.355,332.081,-76.519,-176.584,8.682,148.733
C06860=1157.359,331.833,-76.487,-176.586,8.679,148.733
C06861=1157.363,331.585,-76.454,-176.589,8.675,148.733
C06862=1157.367,331.338,-76.420,-176.592,8.671,148.733
C06863=1157.371,331.089,-76.388,-176.594,8.668,148.732
C06864=1157.375,330.841,-76.355,-176.597,8.665,148.732
C06865=1157.379,330.594,-76.322,-176.599,8.662,148.732
C06866=1157.383,330.346,-76.290,-176.602,8.658,148.732
C06867=1157.387,330.098,-76.257,-176.604,8.654,148.732
C06868=1157.391,329.851,-76.224,-176.606,8.651,148.731
C06869=1157.395,329.602,-76.192,-176.609,8.647,148.731
C06870=1157.399,329.354,-76.158,-176.612,8.644,148.731
C06871=1157.404,329.106,-76.126,-176.614,8.640,148.731
C06872=1157.408,328.859,-76.094,-176.617,8.637,148.731
C06873=1157.412,328.612,-76.061,-176.620,8.633,148.730
C06874=1157.416,328.363,-76.028,-176.622,8.630,148.730
C06875=1157.420,328.116,-75.996,-176.624,8.627,148.730
C06876=1157.424,327.868,-75.963,-176.627,8.623,148.730
C06877=1157.428,327.620,-75.930,-176.629,8.619,148.730
C06878=1157.432,327.372,-75.898,-176.632,8.616,148.729
C06879=1157.436,327.124,-75.865,-176.635,8.612,148.729
C06880=1157.441,326.877,-75.834,-176.637,8.609,148.729
C06881=1157.445,326.628,-75.801,-176.640,8.606,148.729
C06882=1157.449,326.381,-75.768,-176.642,8.602,148.729
C06883=1157.453,326.133,-75.736,-176.645,8.598,148.729
C06884=1157.457,325.885,-75.703,-176.647,8.595,148.728
C06885=1157.461,325.637,-75.671,-176.650,8.592,148.728
C06886=1157.465,325.388,-75.639,-176.653,8.588,148.728
C06887=1157.469,325.142,-75.607,-176.655,8.585,148.728
C06888=1157.474,324.893,-75.574,-176.657,8.581,148.728
C06889=1157.478,324.645,-75.542,-176.660,8.578,148.728
C06890=1157.481,324.398,-75.509,-176.663,8.574,148.727
C06891=1157.486,324.149,-75.477,-176.665,8.571,148.727
C06892=1157.490,323.902,-75.445,-176.668,8.568,148.727
C06893=1157.494,323.654,-75.412,-176.670,8.564,148.727
C06894=1157.498,323.406,-75.380,-176.673,8.560,148.727
C06895=1157.502,323.158,-75.348,-176.675,8.557,148.726
C06896=1157.506,322.910,-75.316,-176.678,8.554,148.726
C06897=1157.510,322.663,-75.284,-176.681,8.550,148.726
C06898=1157.515,322.415,-75.251,-176.683,8.547,148.726
C06899=1157.518,322.167,-75.219,-176.685,8.543,148.726
C06900=1157.523,321.918,-75.187,-176.688,8.540,148.726
C06901=1157.527,321.671,-75.155,-176.691,8.536,148.726
C06902=1157.531,321.423,-75.124,-176.693,8.533,148.725
C06903=1157.535,321.175,-75.090,-176.696,8.530,148.725
C06904=1157.539,320.927,-75.059,-176.698,8.527,148.725
C06905=1157.544,320.680,-75.027,-176.701,8.523,148.725
C06906=1157.547,320.432,-74.995,-176.704,8.519,148.725
C06907=1157.551,320.183,-74.963,-176.706,8.516,148.725
C06908=1157.556,319.936,-74.931,-176.708,8.513,148.724
C06909=1157.560,319.688,-74.899,-176.712,8.509,148.724
C06910=1157.563,319.440,-74.867,-176.714,8.506,148.724
C06911=1157.568,319.191,-74.835,-176.716,8.503,148.724
C06912=1157.572,318.944,-74.803,-176.719,8.499,148.724
C06913=1157.576,318.696,-74.771,-176.721,8.496,148.724
C06914=1157.580,318.448,-74.739,-176.724,8.492,148.724
C06915=1157.585,318.200,-74.707,-176.726,8.489,148.723
C06916=1157.588,317.952,-74.676,-176.729,8.486,148.723
C06917=1157.593,317.704,-74.643,-176.732,8.483,148.723
C06918=1157.597,317.457,-74.612,-176.734,8.479,148.723
C06919=1157.601,317.209,-74.580,-176.737,8.475,148.723
C06920=1157.605,316.961,-74.548,-176.739,8.472,148.723
C06921=1157.610,316.713,-74.516,-176.742,8.469,148.723
C06922=1157.614,316.464,-74.485,-176.745,8.465,148.722
C06923=1157.617,316.216,-74.453,-176.747,8.462,148.722
C06924=1157.622,315.969,-74.421,-176.750,8.459,148.722
C06925=1157.626,315.721,-74.389,-176.752,8.455,148.722
C06926=1157.630,315.473,-74.357,-176.754,8.452,148.722
C06927=1157.634,315.225,-74.326,-176.758,8.448,148.722
C06928=1157.638,314.976,-74.295,-176.760,8.445,148.722
C06929=1157.642,314.729,-74.263,-176.762,8.442,148.721
C06930=1157.646,314.481,-74.231,-176.765,8.439,148.722
C06931=1157.651,314.233,-74.199,-176.767,8.436,148.721
C06932=1157.656,313.955,-74.164,-176.770,8.431,148.721
C06933=1157.661,313.678,-74.129,-176.774,8.428,148.721
C06934=1157.665,313.401,-74.093,-176.776,8.424,148.721
C06935=1157.669,313.123,-74.058,-176.779,8.420,148.721
C06936=1157.674,312.875,-74.027,-176.781,8.417,148.721
C06937=1157.678,312.627,-73.995,-176.784,8.413,148.720
C06938=1157.682,312.380,-73.964,-176.787,8.410,148.720
C06939=1157.686,312.131,-73.933,-176.789,8.407,148.720
C06940=1157.690,311.884,-73.901,-176.792,8.404,148.720
C06941=1157.694,311.635,-73.870,-176.795,8.401,148.720
C06942=1157.699,311.388,-73.838,-176.797,8.397,148.720
C06943=1157.702,311.140,-73.807,-176.800,8.393,148.720
C06944=1157.707,310.892,-73.776,-176.802,8.390,148.720
C06945=1157.711,310.644,-73.744,-176.805,8.387,148.720
C06946=1157.715,310.396,-73.713,-176.807,8.384,148.719
C06947=1157.719,310.148,-73.681,-176.810,8.380,148.719
C06948=1157.724,309.900,-73.651,-176.813,8.377,148.719
C06949=1157.727,309.652,-73.619,-176.815,8.374,148.719
C06950=1157.732,309.404,-73.588,-176.818,8.371,148.719
C06951=1157.736,309.156,-73.556,-176.820,8.367,148.719
C06952=1157.740,308.908,-73.525,-176.823,8.364,148.719
C06953=1157.744,308.660,-73.494,-176.826,8.360,148.719
C06954=1157.749,308.412,-73.463,-176.828,8.357,148.719
C06955=1157.753,308.163,-73.432,-176.831,8.354,148.718
C06956=1157.757,307.916,-73.400,-176.833,8.351,148.718
C06957=1157.761,307.668,-73.369,-176.836,8.348,148.718
C06958=1157.765,307.420,-73.338,-176.839,8.344,148.718
C06959=1157.770,307.172,-73.307,-176.841,8.341,148.718
C06960=1157.774,306.924,-73.276,-176.844,8.337,148.718
C06961=1157.778,306.676,-73.245,-176.846,8.334,148.718
C06962=1157.782,306.428,-73.213,-176.849,8.331,148.718
C06963=1157.787,306.180,-73.182,-176.851,8.328,148.718
C06964=1157.791,305.932,-73.152,-176.854,8.325,148.718
C06965=1157.794,305.684,-73.120,-176.857,8.321,148.717
C06966=1157.799,305.436,-73.090,-176.860,8.318,148.717
C06967=1157.803,305.187,-73.058,-176.862,8.315,148.717
C06968=1157.808,304.939,-73.028,-176.864,8.311,148.717
C06969=1157.812,304.691,-72.997,-176.867,8.308,148.717
C06970=1157.816,304.443,-72.965,-176.869,8.305,148.717
C06971=1157.820,304.196,-72.935,-176.873,8.301,148.717
C06972=1157.824,303.948,-72.904,-176.875,8.298,148.717
C06973=1157.828,303.699,-72.873,-176.878,8.295,148.717
C06974=1157.833,303.451,-72.842,-176.880,8.292,148.716
C06975=1157.838,303.203,-72.811,-176.883,8.289,148.716
C06976=1157.841,302.955,-72.781,-176.885,8.285,148.716
C06977=1157.845,302.707,-72.749,-176.888,8.283,148.716
C06978=1157.850,302.459,-72.719,-176.891,8.278,148.716
C06979=1157.854,302.211,-72.688,-176.893,8.275,148.716
C06980=1157.858,301.963,-72.657,-176.896,8.272,148.716
C06981=1157.862,301.715,-72.627,-176.898,8.269,148.716
C06982=1157.866,301.467,-72.595,-176.901,8.266,148.716
C06983=1157.871,301.219,-72.565,-176.903,8.263,148.716
C06984=1157.875,300.971,-72.535,-176.906,8.260,148.716
C06985=1157.879,300.722,-72.503,-176.908,8.256,148.715
C06986=1157.883,300.474,-72.473,-176.911,8.253,148.715
C06987=1157.887,300.227,-72.442,-176.914,8.249,148.715
C06988=1157.892,299.979,-72.412,-176.917,8.246,148.715
C06989=1157.896,299.730,-72.381,-176.919,8.243,148.715
C06990=1157.900,299.482,-72.351,-176.922,8.240,148.715
C06991=1157.905,299.234,-72.320,-176.924,8.237,148.715
C06992=1157.909,298.986,-72.290,-176.927,8.234,148.715
C06993=1157.913,298.738,-72.259,-176.929,8.231,148.715
C06994=1157.917,298.490,-72.228,-176.932,8.227,148.715
C06995=1157.921,298.242,-72.198,-176.935,8.224,148.715
C06996=1157.926,297.994,-72.167,-176.937,8.221,148.715
C06997=1157.930,297.745,-72.137,-176.940,8.218,148.715
C06998=1157.934,297.497,-72.107,-176.942,8.214,148.715
C06999=1157.939,297.249,-72.076,-176.945,8.211,148.715
C07000=1157.942,297.001,-72.046,-176.947,8.208,148.714
C07001=1157.946,296.753,-72.015,-176.950,8.205,148.714
C07002=1157.951,296.505,-71.985,-176.953,8.202,148.714
C07003=1157.955,296.257,-71.955,-176.956,8.198,148.714
C07004=1157.959,296.009,-71.924,-176.959,8.195,148.714
C07005=1157.964,295.761,-71.894,-176.961,8.192,148.714
C07006=1157.967,295.512,-71.864,-176.964,8.189,148.714
C07007=1157.972,295.264,-71.833,-176.966,8.186,148.714
C07008=1157.976,295.016,-71.803,-176.969,8.183,148.714
C07009=1157.981,294.768,-71.773,-176.971,8.179,148.714
C07010=1157.985,294.520,-71.743,-176.974,8.176,148.714
C07011=1157.989,294.272,-71.712,-176.976,8.173,148.714
C07012=1157.993,294.023,-71.682,-176.979,8.170,148.714
C07013=1157.997,293.775,-71.651,-176.982,8.166,148.714
C07014=1158.002,293.527,-71.622,-176.985,8.163,148.714
C07015=1158.005,293.279,-71.592,-176.987,8.160,148.714
C07016=1158.010,293.031,-71.562,-176.990,8.157,148.713
C07017=1158.014,292.783,-71.531,-176.992,8.154,148.713
C07018=1158.019,292.535,-71.501,-176.995,8.151,148.713
C07019=1158.022,292.286,-71.471,-176.997,8.148,148.713
C07020=1158.026,292.039,-71.441,-177.000,8.145,148.713
C07021=1158.031,291.790,-71.411,-177.003,8.142,148.713
C07022=1158.035,291.542,-71.380,-177.005,8.139,148.713
C07023=1158.039,291.294,-71.351,-177.008,8.136,148.713
C07024=1158.044,291.045,-71.321,-177.010,8.132,148.713
C07025=1158.048,290.798,-71.291,-177.013,8.129,148.713
C07026=1158.052,290.550,-71.261,-177.016,8.126,148.713
C07027=1158.057,290.302,-71.231,-177.019,8.122,148.713
C07028=1158.061,290.053,-71.201,-177.021,8.119,148.713
C07029=1158.065,289.806,-71.171,-177.024,8.116,148.713
C07030=1158.070,289.557,-71.141,-177.027,8.113,148.713
C07031=1158.073,289.308,-71.111,-177.029,8.110,148.713
C07032=1158.077,289.061,-71.081,-177.032,8.107,148.713
C07033=1158.082,288.812,-71.051,-177.034,8.104,148.713
C07034=1158.086,288.564,-71.021,-177.037,8.101,148.713
C07035=1158.090,288.316,-70.991,-177.039,8.098,148.713
C07036=1158.095,288.041,-70.959,-177.043,8.094,148.713
C07037=1158.100,287.766,-70.925,-177.046,8.091,148.713
C07038=1158.105,287.490,-70.893,-177.048,8.087,148.712
C07039=1158.109,287.216,-70.859,-177.051,8.084,148.712
C07040=1158.114,286.967,-70.830,-177.054,8.081,148.712
C07041=1158.118,286.719,-70.801,-177.057,8.078,148.713
C07042=1158.123,286.471,-70.770,-177.059,8.075,148.712
C07043=1158.127,286.222,-70.741,-177.062,8.072,148.712
C07044=1158.131,285.975,-70.711,-177.065,8.069,148.712
C07045=1158.135,285.726,-70.681,-177.067,8.066,148.712
C07046=1158.139,285.478,-70.652,-177.070,8.063,148.712
C07047=1158.143,285.230,-70.622,-177.072,8.060,148.712
C07048=1158.148,284.981,-70.592,-177.075,8.056,148.712
C07049=1158.152,284.733,-70.563,-177.078,8.053,148.712
C07050=1158.157,284.485,-70.534,-177.081,8.050,148.712
C07051=1158.161,284.237,-70.504,-177.083,8.046,148.712
C07052=1158.165,283.989,-70.474,-177.086,8.043,148.712
C07053=1158.169,283.741,-70.444,-177.089,8.040,148.712
C07054=1158.174,283.493,-70.415,-177.091,8.037,148.712
C07055=1158.178,283.245,-70.386,-177.094,8.034,148.712
C07056=1158.182,282.997,-70.356,-177.096,8.031,148.712
C07057=1158.186,282.748,-70.327,-177.099,8.028,148.712
C07058=1158.190,282.500,-70.298,-177.101,8.025,148.712
C07059=1158.195,282.252,-70.268,-177.104,8.022,148.712
C07060=1158.199,282.003,-70.239,-177.107,8.019,148.712
C07061=1158.204,281.754,-70.209,-177.110,8.016,148.712
C07062=1158.208,281.506,-70.180,-177.112,8.013,148.712
C07063=1158.213,281.258,-70.151,-177.115,8.010,148.712
C07064=1158.217,281.010,-70.121,-177.118,8.007,148.712
C07065=1158.221,280.762,-70.092,-177.120,8.004,148.712
C07066=1158.225,280.514,-70.062,-177.123,8.001,148.712
C07067=1158.230,280.265,-70.033,-177.125,7.998,148.712
C07068=1158.233,280.017,-70.004,-177.128,7.995,148.712
C07069=1158.238,279.768,-69.975,-177.131,7.992,148.712
C07070=1158.242,279.521,-69.946,-177.133,7.989,148.712
C07071=1158.247,279.273,-69.917,-177.136,7.986,148.712
C07072=1158.251,279.024,-69.887,-177.139,7.983,148.712
C07073=1158.255,278.776,-69.858,-177.142,7.980,148.712
C07074=1158.259,278.527,-69.829,-177.144,7.976,148.712
C07075=1158.264,278.279,-69.800,-177.147,7.973,148.712
C07076=1158.268,278.031,-69.771,-177.149,7.971,148.712
C07077=1158.273,277.783,-69.741,-177.152,7.968,148.712
C07078=1158.276,277.535,-69.713,-177.154,7.964,148.712
C07079=1158.280,277.286,-69.684,-177.157,7.961,148.712
C07080=1158.285,277.038,-69.654,-177.160,7.958,148.712
C07081=1158.290,276.790,-69.626,-177.163,7.955,148.712
C07082=1158.294,276.542,-69.596,-177.166,7.952,148.712
C07083=1158.298,276.293,-69.567,-177.168,7.949,148.712
C07084=1158.302,276.045,-69.539,-177.171,7.946,148.712
C07085=1158.306,275.796,-69.509,-177.173,7.943,148.712
C07086=1158.311,275.549,-69.480,-177.176,7.940,148.712
C07087=1158.315,275.300,-69.451,-177.179,7.937,148.712
C07088=1158.319,275.052,-69.422,-177.181,7.934,148.712
C07089=1158.323,274.803,-69.394,-177.184,7.931,148.712
C07090=1158.328,274.556,-69.365,-177.187,7.928,148.712
C07091=1158.332,274.307,-69.336,-177.189,7.925,148.712
C07092=1158.337,274.058,-69.307,-177.192,7.922,148.712
C07093=1158.341,273.811,-69.279,-177.195,7.919,148.712
C07094=1158.345,273.562,-69.249,-177.197,7.916,148.712
C07095=1158.350,273.313,-69.221,-177.200,7.913,148.712
C07096=1158.354,273.065,-69.191,-177.203,7.910,148.712
C07097=1158.358,272.817,-69.163,-177.206,7.907,148.712
C07098=1158.362,272.569,-69.134,-177.208,7.904,148.712
C07099=1158.367,272.320,-69.105,-177.211,7.901,148.712
C07100=1158.371,272.073,-69.077,-177.213,7.898,148.712
C07101=1158.375,271.824,-69.048,-177.216,7.896,148.712
C07102=1158.380,271.575,-69.019,-177.218,7.893,148.712
C07103=1158.384,271.328,-68.991,-177.221,7.890,148.712
C07104=1158.388,271.079,-68.962,-177.224,7.887,148.712
C07105=1158.393,270.831,-68.933,-177.227,7.884,148.712
C07106=1158.397,270.583,-68.905,-177.229,7.881,148.712
C07107=1158.401,270.334,-68.876,-177.232,7.878,148.712
C07108=1158.406,270.085,-68.847,-177.234,7.875,148.712
C07109=1158.410,269.838,-68.819,-177.237,7.872,148.712
C07110=1158.414,269.589,-68.790,-177.240,7.869,148.712
C07111=1158.418,269.340,-68.762,-177.243,7.866,148.712
C07112=1158.423,269.093,-68.733,-177.246,7.863,148.712
C07113=1158.427,268.844,-68.705,-177.248,7.860,148.712
C07114=1158.432,268.596,-68.676,-177.251,7.857,148.712
C07115=1158.436,268.347,-68.648,-177.253,7.854,148.712
C07116=1158.440,268.098,-68.619,-177.256,7.851,148.712
C07117=1158.445,267.851,-68.590,-177.259,7.848,148.712
C07118=1158.449,267.602,-68.562,-177.262,7.845,148.713
C07119=1158.454,267.354,-68.534,-177.264,7.842,148.713
C07120=1158.457,267.106,-68.506,-177.267,7.840,148.713
C07121=1158.463,266.857,-68.477,-177.269,7.837,148.713
C07122=1158.466,266.609,-68.449,-177.272,7.834,148.713
C07123=1158.471,266.360,-68.420,-177.274,7.831,148.713
C07124=1158.475,266.113,-68.392,-177.277,7.828,148.713
C07125=1158.479,265.864,-68.363,-177.280,7.825,148.713
C07126=1158.484,265.616,-68.335,-177.283,7.822,148.713
C07127=1158.488,265.367,-68.307,-177.286,7.819,148.713
C07128=1158.492,265.119,-68.279,-177.288,7.816,148.713
C07129=1158.496,264.871,-68.251,-177.291,7.813,148.713
C07130=1158.501,264.622,-68.222,-177.294,7.810,148.713
C07131=1158.505,264.374,-68.194,-177.297,7.807,148.713
C07132=1158.510,264.126,-68.166,-177.299,7.804,148.713
C07133=1158.514,263.877,-68.138,-177.302,7.802,148.713
C07134=1158.519,263.629,-68.109,-177.304,7.799,148.713
C07135=1158.523,263.380,-68.081,-177.307,7.796,148.713
C07136=1158.527,263.132,-68.053,-177.310,7.793,148.713
C07137=1158.532,262.884,-68.025,-177.313,7.790,148.713
C07138=1158.536,262.635,-67.998,-177.315,7.787,148.713
C07139=1158.540,262.386,-67.969,-177.318,7.784,148.713
C07140=1158.545,262.113,-67.937,-177.320,7.781,148.713
C07141=1158.550,261.840,-67.907,-177.324,7.779,148.714
C07142=1158.554,261.567,-67.876,-177.327,7.775,148.714
C07143=1158.560,261.294,-67.846,-177.330,7.772,148.714
C07144=1158.563,261.046,-67.818,-177.333,7.769,148.714
C07145=1158.569,260.797,-67.789,-177.335,7.766,148.714
C07146=1158.573,260.548,-67.762,-177.338,7.763,148.714
C07147=1158.577,260.300,-67.734,-177.341,7.760,148.714
C07148=1158.581,260.052,-67.706,-177.344,7.757,148.714
C07149=1158.586,259.804,-67.678,-177.345,7.755,148.714
C07150=1158.590,259.555,-67.651,-177.348,7.752,148.714
C07151=1158.594,259.306,-67.622,-177.351,7.749,148.714
C07152=1158.599,259.059,-67.595,-177.354,7.746,148.714
C07153=1158.603,258.810,-67.566,-177.356,7.743,148.714
C07154=1158.608,258.561,-67.539,-177.359,7.740,148.714
C07155=1158.612,258.313,-67.511,-177.362,7.737,148.714
C07156=1158.616,258.065,-67.483,-177.365,7.734,148.714
C07157=1158.620,257.816,-67.456,-177.367,7.732,148.714
C07158=1158.625,257.567,-67.427,-177.370,7.729,148.714
C07159=1158.630,257.319,-67.400,-177.372,7.726,148.715
C07160=1158.634,257.071,-67.372,-177.375,7.723,148.715
C07161=1158.638,256.822,-67.344,-177.378,7.720,148.715
C07162=1158.642,256.574,-67.317,-177.381,7.718,148.715
C07163=1158.647,256.326,-67.289,-177.384,7.715,148.715
C07164=1158.651,256.077,-67.262,-177.387,7.712,148.715
C07165=1158.656,255.829,-67.233,-177.389,7.710,148.715
C07166=1158.660,255.580,-67.206,-177.392,7.707,148.715
C07167=1158.664,255.332,-67.178,-177.394,7.704,148.715
C07168=1158.669,255.083,-67.151,-177.397,7.701,148.715
C07169=1158.673,254.835,-67.123,-177.400,7.698,148.715
C07170=1158.677,254.586,-67.096,-177.403,7.695,148.715
C07171=1158.682,254.338,-67.068,-177.406,7.692,148.716
C07172=1158.686,254.090,-67.041,-177.408,7.690,148.716
C07173=1158.690,253.841,-67.013,-177.411,7.687,148.716
C07174=1158.695,253.593,-66.986,-177.413,7.684,148.716
C07175=1158.699,253.345,-66.958,-177.416,7.681,148.716
C07176=1158.704,253.096,-66.931,-177.419,7.678,148.716
C07177=1158.708,252.847,-66.904,-177.422,7.675,148.716
C07178=1158.712,252.599,-66.876,-177.424,7.673,148.716
C07179=1158.717,252.351,-66.849,-177.427,7.670,148.716
C07180=1158.721,252.102,-66.822,-177.429,7.667,148.716
C07181=1158.725,251.854,-66.794,-177.432,7.664,148.716
C07182=1158.730,251.605,-66.767,-177.435,7.661,148.716
C07183=1158.735,251.357,-66.740,-177.438,7.658,148.717
C07184=1158.739,251.109,-66.712,-177.440,7.656,148.717
C07185=1158.743,250.860,-66.684,-177.443,7.653,148.717
C07186=1158.748,250.611,-66.657,-177.446,7.650,148.717
C07187=1158.752,250.363,-66.629,-177.449,7.648,148.717
C07188=1158.757,250.115,-66.602,-177.451,7.645,148.717
C07189=1158.761,249.865,-66.575,-177.454,7.642,148.717
C07190=1158.765,249.617,-66.548,-177.456,7.639,148.717
C07191=1158.770,249.368,-66.521,-177.459,7.637,148.717
C07192=1158.774,249.121,-66.494,-177.462,7.634,148.717
C07193=1158.778,248.872,-66.467,-177.465,7.631,148.717
C07194=1158.782,248.623,-66.439,-177.468,7.628,148.718
C07195=1158.787,248.375,-66.412,-177.471,7.625,148.718
C07196=1158.792,248.126,-66.385,-177.473,7.623,148.718
C07197=1158.796,247.878,-66.358,-177.476,7.620,148.718
C07198=1158.801,247.629,-66.331,-177.478,7.617,148.718
C07199=1158.805,247.382,-66.304,-177.481,7.614,148.718
C07200=1158.809,247.133,-66.277,-177.484,7.611,148.718
C07201=1158.813,246.884,-66.249,-177.486,7.609,148.718
C07202=1158.818,246.635,-66.222,-177.489,7.606,148.718
C07203=1158.823,246.387,-66.195,-177.492,7.604,148.719
C07204=1158.826,246.139,-66.169,-177.495,7.601,148.719
C07205=1158.831,245.890,-66.142,-177.498,7.598,148.719
C07206=1158.836,245.642,-66.115,-177.500,7.596,148.719
C07207=1158.840,245.393,-66.088,-177.503,7.593,148.719
C07208=1158.844,245.144,-66.061,-177.505,7.590,148.719
C07209=1158.848,244.896,-66.034,-177.509,7.587,148.719
C07210=1158.853,244.647,-66.007,-177.511,7.584,148.719
C07211=1158.858,244.399,-65.979,-177.514,7.582,148.719
C07212=1158.862,244.151,-65.953,-177.516,7.579,148.719
C07213=1158.866,243.902,-65.926,-177.519,7.576,148.720
C07214=1158.871,243.653,-65.900,-177.522,7.573,148.720
C07215=1158.875,243.405,-65.873,-177.524,7.571,148.720
C07216=1158.880,243.156,-65.846,-177.527,7.568,148.720
C07217=1158.884,242.908,-65.819,-177.530,7.565,148.720
C07218=1158.888,242.660,-65.793,-177.533,7.563,148.720
C07219=1158.893,242.411,-65.765,-177.536,7.560,148.720
C07220=1158.898,242.163,-65.738,-177.538,7.557,148.720
C07221=1158.902,241.914,-65.713,-177.541,7.555,148.720
C07222=1158.906,241.665,-65.685,-177.544,7.552,148.721
C07223=1158.911,241.416,-65.658,-177.547,7.549,148.721
C07224=1158.915,241.168,-65.632,-177.549,7.547,148.721
C07225=1158.919,240.920,-65.605,-177.552,7.544,148.721
C07226=1158.923,240.671,-65.579,-177.554,7.541,148.721
C07227=1158.928,240.422,-65.552,-177.558,7.538,148.721
C07228=1158.933,240.174,-65.525,-177.560,7.536,148.721
C07229=1158.937,239.925,-65.499,-177.563,7.533,148.721
C07230=1158.942,239.676,-65.472,-177.565,7.530,148.722
C07231=1158.946,239.428,-65.446,-177.568,7.527,148.722
C07232=1158.951,239.179,-65.419,-177.571,7.526,148.722
C07233=1158.954,238.931,-65.393,-177.574,7.523,148.722
C07234=1158.959,238.683,-65.366,-177.576,7.520,148.722
C07235=1158.964,238.434,-65.340,-177.579,7.517,148.722
C07236=1158.969,238.186,-65.313,-177.581,7.515,148.722
C07237=1158.973,237.938,-65.287,-177.585,7.512,148.723
C07238=1158.977,237.689,-65.260,-177.587,7.509,148.723
C07239=1158.981,237.440,-65.234,-177.590,7.506,148.723
C07240=1158.986,237.191,-65.208,-177.592,7.504,148.723
C07241=1158.990,236.943,-65.181,-177.596,7.501,148.723
C07242=1158.995,236.694,-65.155,-177.598,7.499,148.723
C07243=1158.999,236.446,-65.128,-177.601,7.496,148.723
C07244=1159.004,236.174,-65.099,-177.604,7.493,148.723
C07245=1159.009,235.902,-65.071,-177.607,7.490,148.724
C07246=1159.014,235.631,-65.042,-177.610,7.487,148.724
C07247=1159.019,235.359,-65.014,-177.613,7.484,148.724
C07248=1159.023,235.110,-64.986,-177.616,7.482,148.724
C07249=1159.028,234.862,-64.961,-177.618,7.479,148.724
C07250=1159.032,234.613,-64.934,-177.621,7.477,148.724
C07251=1159.037,234.364,-64.908,-177.624,7.474,148.724
C07252=1159.041,234.115,-64.882,-177.626,7.472,148.725
C07253=1159.045,233.867,-64.855,-177.629,7.469,148.725
C07254=1159.050,233.619,-64.830,-177.632,7.466,148.725
C07255=1159.054,233.371,-64.803,-177.635,7.463,148.725
C07256=1159.059,233.122,-64.777,-177.637,7.461,148.725
C07257=1159.063,232.873,-64.751,-177.640,7.458,148.725
C07258=1159.067,232.625,-64.725,-177.643,7.455,148.725
C07259=1159.072,232.375,-64.698,-177.645,7.454,148.726
C07260=1159.077,232.127,-64.673,-177.648,7.451,148.726
C07261=1159.081,231.879,-64.646,-177.651,7.448,148.726
C07262=1159.085,231.630,-64.621,-177.653,7.446,148.726
C07263=1159.090,231.381,-64.594,-177.656,7.443,148.726
C07264=1159.094,231.132,-64.569,-177.659,7.440,148.726
C07265=1159.098,230.884,-64.542,-177.662,7.437,148.726
C07266=1159.104,230.636,-64.516,-177.665,7.435,148.727
C07267=1159.108,230.387,-64.490,-177.667,7.432,148.727
C07268=1159.112,230.138,-64.465,-177.670,7.429,148.727
C07269=1159.117,229.889,-64.439,-177.672,7.427,148.727
C07270=1159.120,229.641,-64.412,-177.676,7.425,148.727
C07271=1159.126,229.393,-64.386,-177.678,7.422,148.727
C07272=1159.130,229.144,-64.361,-177.681,7.420,148.728
C07273=1159.134,228.895,-64.335,-177.684,7.417,148.728
C07274=1159.139,228.646,-64.309,-177.687,7.414,148.728
C07275=1159.144,228.398,-64.284,-177.689,7.412,148.728
C07276=1159.149,228.149,-64.257,-177.692,7.409,148.728
C07277=1159.153,227.900,-64.232,-177.695,7.406,148.728
C07278=1159.157,227.652,-64.205,-177.697,7.404,148.729
C07279=1159.161,227.404,-64.180,-177.700,7.402,148.729
C07280=1159.166,227.155,-64.154,-177.703,7.399,148.729
C07281=1159.170,226.906,-64.128,-177.705,7.397,148.729
C07282=1159.174,226.658,-64.103,-177.709,7.394,148.729
C07283=1159.180,226.409,-64.077,-177.711,7.391,148.729
C07284=1159.184,226.160,-64.051,-177.714,7.389,148.730
C07285=1159.188,225.912,-64.025,-177.717,7.386,148.730
C07286=1159.193,225.664,-64.000,-177.720,7.383,148.730
C07287=1159.197,225.415,-63.974,-177.722,7.381,148.730
C07288=1159.201,225.166,-63.948,-177.725,7.379,148.730
C07289=1159.207,224.917,-63.924,-177.728,7.376,148.730
C07290=1159.211,224.668,-63.898,-177.730,7.374,148.731
C07291=1159.215,224.420,-63.872,-177.733,7.371,148.731
C07292=1159.220,224.171,-63.847,-177.735,7.369,148.731
C07293=1159.224,223.923,-63.821,-177.738,7.366,148.731
C07294=1159.228,223.674,-63.795,-177.741,7.363,148.731
C07295=1159.233,223.426,-63.770,-177.744,7.361,148.731
C07296=1159.237,223.177,-63.744,-177.746,7.358,148.732
C07297=1159.242,222.928,-63.719,-177.750,7.356,148.732
C07298=1159.247,222.679,-63.694,-177.752,7.354,148.732
C07299=1159.251,222.431,-63.668,-177.755,7.351,148.732
C07300=1159.255,222.182,-63.642,-177.757,7.349,148.732
C07301=1159.260,221.934,-63.617,-177.760,7.346,148.733
C07302=1159.265,221.684,-63.592,-177.763,7.343,148.733
C07303=1159.269,221.436,-63.566,-177.766,7.341,148.733
C07304=1159.274,221.187,-63.541,-177.768,7.338,148.733
C07305=1159.278,220.939,-63.515,-177.772,7.336,148.733
C07306=1159.283,220.690,-63.490,-177.774,7.334,148.733
C07307=1159.287,220.441,-63.464,-177.777,7.331,148.734
C07308=1159.292,220.193,-63.439,-177.779,7.329,148.734
C07309=1159.296,219.944,-63.414,-177.782,7.326,148.734
C07310=1159.300,219.695,-63.389,-177.785,7.323,148.734
C07311=1159.305,219.447,-63.363,-177.787,7.321,148.734
C07312=1159.309,219.198,-63.338,-177.791,7.319,148.735
C07313=1159.314,218.949,-63.313,-177.793,7.317,148.735
C07314=1159.318,218.701,-63.287,-177.796,7.314,148.735
